LIN {X -0.158,Y -481.515,Z 1004.070,A 0.000,B 0.000,C 90.000,E1 228.528} C_DIS
LIN {X -0.055,Y -475.509,Z 1004.054,A 0.000,B 0.000,C 90.000,E1 225.729} C_DIS
LIN {X -0.116,Y -471.668,Z 1004.044,A 0.000,B 0.000,C 90.000,E1 223.866} C_DIS
LIN {X -0.012,Y -468.320,Z 1004.035,A 0.000,B 0.000,C 90.000,E1 222.285} C_DIS
LIN {X 0.118,Y -464.188,Z 1004.024,A 0.000,B 0.000,C 90.000,E1 220.378} C_DIS
LIN {X 0.208,Y -459.845,Z 1004.014,A 0.000,B 0.000,C 90.000,E1 218.463} C_DIS
LIN {X -0.083,Y -455.698,Z 1004.003,A 0.000,B 0.000,C 90.000,E1 216.583} C_DIS
LIN {X 0.261,Y -451.461,Z 1003.992,A 0.000,B 0.000,C 90.000,E1 214.612} C_DIS
LIN {X 0.003,Y -447.260,Z 1003.982,A 0.000,B 0.000,C 90.000,E1 212.704} C_DIS
LIN {X -0.029,Y -443.708,Z 1003.973,A 0.000,B 0.000,C 90.000,E1 211.082} C_DIS
LIN {X -0.140,Y -440.143,Z 1003.964,A 0.000,B 0.000,C 90.000,E1 209.461} C_DIS
LIN {X 0.041,Y -435.600,Z 1003.953,A 0.000,B 0.000,C 90.000,E1 207.462} C_DIS
LIN {X 0.115,Y -431.912,Z 1003.943,A 0.000,B 0.000,C 90.000,E1 205.796} C_DIS
LIN {X 0.105,Y -428.119,Z 1003.934,A 0.000,B 0.000,C 90.000,E1 204.131} C_DIS
LIN {X -0.147,Y -423.631,Z 1003.923,A 0.000,B 0.000,C 90.000,E1 202.153} C_DIS
LIN {X -0.164,Y -417.964,Z 1003.908,A 0.000,B 0.000,C 90.000,E1 199.450} C_DIS
LIN {X -0.090,Y -411.609,Z 1003.889,A 0.000,B 0.000,C 90.000,E1 196.024} C_DIS
LIN {X -0.066,Y -408.697,Z 1003.879,A 0.000,B 0.000,C 90.000,E1 194.300} C_DIS
LIN {X 0.193,Y -405.963,Z 1003.870,A 0.000,B 0.000,C 90.000,E1 192.535} C_DIS
LIN {X -0.085,Y -403.341,Z 1003.860,A 0.000,B 0.000,C 90.000,E1 190.838} C_DIS
LIN {X -0.083,Y -401.810,Z 1003.854,A 0.000,B 0.000,C 90.000,E1 189.792} C_DIS
LIN {X -0.106,Y -400.288,Z 1003.847,A 0.000,B 0.000,C 90.000,E1 188.398} C_DIS
LIN {X -0.144,Y -400.025,Z 1003.841,A 0.000,B 0.000,C 90.000,E1 187.352} C_DIS
LIN {X -0.116,Y -400.167,Z 1003.839,A 0.000,B 0.000,C 90.000,E1 187.004} C_DIS
LIN {X 0.119,Y -400.532,Z 1003.838,A 0.000,B 0.000,C 90.000,E1 186.777} C_DIS
LIN {X 0.045,Y -401.446,Z 1003.834,A 0.000,B 0.000,C 90.000,E1 186.087} C_DIS
LIN {X 0.019,Y -402.755,Z 1003.831,A 0.000,B 0.000,C 90.000,E1 185.568} C_DIS
LIN {X 0.143,Y -405.533,Z 1003.827,A 0.000,B 0.000,C 90.000,E1 184.878} C_DIS
LIN {X 0.140,Y -407.318,Z 1003.825,A 0.000,B 0.000,C 90.000,E1 184.531} C_DIS
LIN {X 0.080,Y -410.355,Z 1003.823,A 0.000,B 0.000,C 90.000,E1 184.073} C_DIS
LIN {X 0.140,Y -415.263,Z 1003.819,A 0.000,B 0.000,C 90.000,E1 183.440} C_DIS
LIN {X -0.203,Y -423.575,Z 1003.814,A 0.000,B 0.000,C 90.000,E1 182.522} C_DIS
LIN {X -0.028,Y -430.671,Z 1003.810,A 0.000,B 0.000,C 90.000,E1 181.718} C_DIS
LIN {X 0.109,Y -442.868,Z 1003.802,A 0.000,B 0.000,C 90.000,E1 180.344} C_DIS
LIN {X 0.157,Y -455.130,Z 1003.794,A 0.000,B 0.000,C 90.000,E1 178.969} C_DIS
LIN {X 0.082,Y -463.200,Z 1003.789,A 0.000,B 0.000,C 90.000,E1 178.051} C_DIS
LIN {X 0.169,Y -468.505,Z 1003.786,A 0.000,B 0.000,C 90.000,E1 177.421} C_DIS
LIN {X 0.143,Y -476.033,Z 1003.781,A 0.000,B 0.000,C 90.000,E1 176.502} C_DIS
LIN {X -0.110,Y -482.206,Z 1003.776,A 0.000,B 0.000,C 90.000,E1 175.755} C_DIS
LIN {X 0.000,Y -490.150,Z 1003.770,A 0.000,B 0.000,C 90.000,E1 174.666} C_DIS
LIN {X 0.089,Y -496.507,Z 1003.765,A 0.000,B 0.000,C 90.000,E1 173.742} C_DIS
LIN {X 0.009,Y -503.705,Z 1003.760,A 0.000,B 0.000,C 90.000,E1 172.704} C_DIS
LIN {X -0.213,Y -511.598,Z 1003.753,A 0.000,B 0.000,C 90.000,E1 171.546} C_DIS
LIN {X -0.104,Y -519.992,Z 1003.746,A 0.000,B 0.000,C 90.000,E1 170.208} C_DIS
LIN {X 0.120,Y -526.038,Z 1003.740,A 0.000,B 0.000,C 90.000,E1 169.162} C_DIS
LIN {X -0.160,Y -528.740,Z 1003.737,A 0.000,B 0.000,C 90.000,E1 168.757} C_DIS
LIN {X 0.215,Y -538.987,Z 1003.728,A 0.000,B 0.000,C 90.000,E1 166.992} C_DIS
LIN {X 0.272,Y -544.731,Z 1003.722,A 0.000,B 0.000,C 90.000,E1 165.992} C_DIS
LIN {X 0.014,Y -549.638,Z 1003.718,A 0.000,B 0.000,C 90.000,E1 165.172} C_DIS
LIN {X -0.192,Y -555.149,Z 1003.712,A 0.000,B 0.000,C 90.000,E1 164.212} C_DIS
LIN {X -0.191,Y -561.923,Z 1003.705,A 0.000,B 0.000,C 90.000,E1 162.960} C_DIS
LIN {X 0.244,Y -569.849,Z 1003.697,A 0.000,B 0.000,C 90.000,E1 161.402} C_DIS
LIN {X -0.065,Y -574.593,Z 1003.692,A 0.000,B 0.000,C 90.000,E1 160.477} C_DIS
LIN {X 0.112,Y -578.574,Z 1003.687,A 0.000,B 0.000,C 90.000,E1 159.645} C_DIS
LIN {X -0.089,Y -582.935,Z 1003.682,A 0.000,B 0.000,C 90.000,E1 158.720} C_DIS
LIN {X 0.111,Y -586.015,Z 1003.678,A 0.000,B 0.000,C 90.000,E1 158.028} C_DIS
LIN {X -0.060,Y -590.629,Z 1003.672,A 0.000,B 0.000,C 90.000,E1 156.975} C_DIS
LIN {X -0.174,Y -594.836,Z 1003.666,A 0.000,B 0.000,C 90.000,E1 155.921} C_DIS
LIN {X 0.009,Y -598.632,Z 1003.660,A 0.000,B 0.000,C 90.000,E1 154.845} C_DIS
LIN {X 0.319,Y -601.320,Z 1003.656,A 0.000,B 0.000,C 90.000,E1 154.024} C_DIS
LIN {X 0.052,Y -604.541,Z 1003.650,A 0.000,B 0.000,C 90.000,E1 152.999} C_DIS
LIN {X 0.011,Y -609.120,Z 1003.641,A 0.000,B 0.000,C 90.000,E1 151.435} C_DIS
LIN {X 0.062,Y -613.469,Z 1003.633,A 0.000,B 0.000,C 90.000,E1 149.871} C_DIS
LIN {X -0.290,Y -616.337,Z 1003.627,A 0.000,B 0.000,C 90.000,E1 148.869} C_DIS
LIN {X 0.222,Y -619.799,Z 1003.620,A 0.000,B 0.000,C 90.000,E1 147.533} C_DIS
LIN {X 0.054,Y -624.612,Z 1003.610,A 0.000,B 0.000,C 90.000,E1 145.754} C_DIS
LIN {X -0.164,Y -629.479,Z 1003.600,A 0.000,B 0.000,C 90.000,E1 143.989} C_DIS
LIN {X -0.261,Y -633.516,Z 1003.591,A 0.000,B 0.000,C 90.000,E1 142.477} C_DIS
LIN {X 0.234,Y -636.871,Z 1003.584,A 0.000,B 0.000,C 90.000,E1 141.170} C_DIS
LIN {X 0.289,Y -640.156,Z 1003.577,A 0.000,B 0.000,C 90.000,E1 139.908} C_DIS
LIN {X -0.007,Y -642.774,Z 1003.572,A 0.000,B 0.000,C 90.000,E1 138.933} C_DIS
LIN {X -0.084,Y -647.947,Z 1003.561,A 0.000,B 0.000,C 90.000,E1 136.944} C_DIS
LIN {X 0.037,Y -652.110,Z 1003.553,A 0.000,B 0.000,C 90.000,E1 135.445} C_DIS
LIN {X 0.114,Y -659.741,Z 1003.539,A 0.000,B 0.000,C 90.000,E1 132.975} C_DIS
LIN {X 0.065,Y -666.201,Z 1003.528,A 0.000,B 0.000,C 90.000,E1 131.024} C_DIS
LIN {X -0.397,Y -669.403,Z 1003.523,A 0.000,B 0.000,C 90.000,E1 130.092} C_DIS
LIN {X -0.316,Y -672.466,Z 1003.517,A 0.000,B 0.000,C 90.000,E1 129.116} C_DIS
LIN {X -0.082,Y -675.979,Z 1003.510,A 0.000,B 0.000,C 90.000,E1 127.890} C_DIS
LIN {X -0.176,Y -680.134,Z 1003.503,A 0.000,B 0.000,C 90.000,E1 126.457} C_DIS
LIN {X -0.198,Y -684.071,Z 1003.495,A 0.000,B 0.000,C 90.000,E1 125.025} C_DIS
LIN {X -0.181,Y -687.276,Z 1003.488,A 0.000,B 0.000,C 90.000,E1 123.833} C_DIS
LIN {X 0.235,Y -689.124,Z 1003.484,A 0.000,B 0.000,C 90.000,E1 123.086} C_DIS
LIN {X 0.178,Y -692.714,Z 1003.476,A 0.000,B 0.000,C 90.000,E1 121.671} C_DIS
LIN {X -0.059,Y -695.075,Z 1003.471,A 0.000,B 0.000,C 90.000,E1 120.747} C_DIS
LIN {X -0.166,Y -696.680,Z 1003.467,A 0.000,B 0.000,C 90.000,E1 120.050} C_DIS
LIN {X 0.341,Y -697.649,Z 1003.464,A 0.000,B 0.000,C 90.000,E1 119.539} C_DIS
LIN {X 0.163,Y -699.184,Z 1003.459,A 0.000,B 0.000,C 90.000,E1 118.615} C_DIS
LIN {X -0.328,Y -700.404,Z 1003.454,A 0.000,B 0.000,C 90.000,E1 117.719} C_DIS
LIN {X -0.324,Y -701.880,Z 1003.443,A 0.000,B 0.000,C 90.000,E1 115.848} C_DIS
LIN {X -0.149,Y -702.550,Z 1003.438,A 0.000,B 0.000,C 90.000,E1 114.899} C_DIS
LIN {X -0.244,Y -702.705,Z 1003.434,A 0.000,B 0.000,C 90.000,E1 114.207} C_DIS
LIN {X 0.310,Y -702.127,Z 1003.432,A 0.000,B 0.000,C 90.000,E1 113.695} C_DIS
LIN {X -0.339,Y -701.687,Z 1003.431,A 0.000,B 0.000,C 90.000,E1 113.515} C_DIS
LIN {X 0.065,Y -699.072,Z 1003.427,A 0.000,B 0.000,C 90.000,E1 112.898} C_DIS
LIN {X 0.199,Y -698.300,Z 1003.427,A 0.000,B 0.000,C 90.000,E1 112.770} C_DIS
LIN {X 0.328,Y -697.150,Z 1003.426,A 0.000,B 0.000,C 90.000,E1 112.642} C_DIS
LIN {X 0.151,Y -692.817,Z 1003.424,A 0.000,B 0.000,C 90.000,E1 112.333} C_DIS
LIN {X -0.159,Y -691.331,Z 1003.424,A 0.000,B 0.000,C 90.000,E1 112.259} C_DIS
LIN {X -0.092,Y -689.495,Z 1003.423,A 0.000,B 0.000,C 90.000,E1 112.153} C_DIS
LIN {X 0.058,Y -684.547,Z 1003.422,A 0.000,B 0.000,C 90.000,E1 111.972} C_DIS
LIN {X 0.216,Y -677.312,Z 1003.422,A 0.000,B 0.000,C 90.000,E1 111.844} C_DIS
LIN {X -0.113,Y -675.141,Z 1003.421,A 0.000,B 0.000,C 90.000,E1 111.844} C_DIS
LIN {X -0.164,Y -669.455,Z 1003.421,A 0.000,B 0.000,C 90.000,E1 111.844} C_DIS
LIN {X -0.198,Y -618.340,Z 1003.421,A 0.000,B 0.000,C 90.000,E1 111.844} C_DIS
LIN {X -0.208,Y -614.996,Z 1003.421,A 0.000,B 0.000,C 90.000,E1 111.770} C_DIS
LIN {X -0.025,Y -610.858,Z 1003.420,A 0.000,B 0.000,C 90.000,E1 111.642} C_DIS
LIN {X -0.146,Y -604.502,Z 1003.419,A 0.000,B 0.000,C 90.000,E1 111.408} C_DIS
LIN {X -0.108,Y -601.661,Z 1003.418,A 0.000,B 0.000,C 90.000,E1 111.280} C_DIS
LIN {X -0.047,Y -595.162,Z 1003.416,A 0.000,B 0.000,C 90.000,E1 110.918} C_DIS
LIN {X 0.031,Y -589.063,Z 1003.414,A 0.000,B 0.000,C 90.000,E1 110.482} C_DIS
LIN {X 0.107,Y -577.100,Z 1003.408,A 0.000,B 0.000,C 90.000,E1 109.504} C_DIS
LIN {X 0.298,Y -572.724,Z 1003.407,A 0.000,B 0.000,C 90.000,E1 109.141} C_DIS
LIN {X -0.084,Y -564.162,Z 1003.404,A 0.000,B 0.000,C 90.000,E1 108.671} C_DIS
LIN {X 0.140,Y -550.287,Z 1003.400,A 0.000,B 0.000,C 90.000,E1 107.946} C_DIS
LIN {X -0.224,Y -548.864,Z 1003.399,A 0.000,B 0.000,C 90.000,E1 107.819} C_DIS
LIN {X -0.266,Y -548.850,Z 1003.399,A 0.000,B 0.000,C 90.000,E1 107.819} C_DIS
LIN {X -0.134,Y -548.453,Z 1003.397,A 0.000,B 0.000,C 90.000,E1 107.511} C_DIS
LIN {X -0.090,Y -548.522,Z 1003.393,A 0.000,B 0.000,C 90.000,E1 106.804} C_DIS
LIN {X 0.171,Y -549.154,Z 1003.386,A 0.000,B 0.000,C 90.000,E1 105.371} C_DIS
LIN {X 0.220,Y -550.329,Z 1003.373,A 0.000,B 0.000,C 90.000,E1 103.119} C_DIS
LIN {X 0.288,Y -552.781,Z 1003.357,A 0.000,B 0.000,C 90.000,E1 100.310} C_DIS
LIN {X -0.130,Y -554.939,Z 1003.347,A 0.000,B 0.000,C 90.000,E1 98.398} C_DIS
LIN {X -0.133,Y -556.428,Z 1003.339,A 0.000,B 0.000,C 90.000,E1 97.004} C_DIS
LIN {X -0.246,Y -557.751,Z 1003.331,A 0.000,B 0.000,C 90.000,E1 95.625} C_DIS
LIN {X 0.230,Y -558.784,Z 1003.323,A 0.000,B 0.000,C 90.000,E1 94.188} C_DIS
LIN {X 0.162,Y -559.630,Z 1003.316,A 0.000,B 0.000,C 90.000,E1 92.808} C_DIS
LIN {X -0.209,Y -560.695,Z 1003.303,A 0.000,B 0.000,C 90.000,E1 90.630} C_DIS
LIN {X 0.174,Y -561.210,Z 1003.297,A 0.000,B 0.000,C 90.000,E1 89.484} C_DIS
LIN {X 0.115,Y -561.773,Z 1003.290,A 0.000,B 0.000,C 90.000,E1 88.108} C_DIS
LIN {X 0.069,Y -562.004,Z 1003.282,A 0.000,B 0.000,C 90.000,E1 86.731} C_DIS
LIN {X -0.073,Y -562.162,Z 1003.276,A 0.000,B 0.000,C 90.000,E1 85.641} C_DIS
LIN {X -0.082,Y -562.395,Z 1003.268,A 0.000,B 0.000,C 90.000,E1 84.261} C_DIS
LIN {X 0.204,Y -562.712,Z 1003.257,A 0.000,B 0.000,C 90.000,E1 82.299} C_DIS
LIN {X -0.142,Y -563.152,Z 1003.248,A 0.000,B 0.000,C 90.000,E1 80.679} C_DIS
LIN {X -0.228,Y -563.904,Z 1003.237,A 0.000,B 0.000,C 90.000,E1 78.757} C_DIS
LIN {X 0.201,Y -564.750,Z 1003.228,A 0.000,B 0.000,C 90.000,E1 77.061} C_DIS
LIN {X 0.221,Y -565.722,Z 1003.219,A 0.000,B 0.000,C 90.000,E1 75.408} C_DIS
LIN {X -0.129,Y -566.892,Z 1003.210,A 0.000,B 0.000,C 90.000,E1 73.795} C_DIS
LIN {X -0.116,Y -568.379,Z 1003.199,A 0.000,B 0.000,C 90.000,E1 71.873} C_DIS
LIN {X 0.110,Y -569.709,Z 1003.189,A 0.000,B 0.000,C 90.000,E1 69.934} C_DIS
LIN {X 0.206,Y -570.687,Z 1003.180,A 0.000,B 0.000,C 90.000,E1 68.284} C_DIS
LIN {X 0.171,Y -571.364,Z 1003.172,A 0.000,B 0.000,C 90.000,E1 66.922} C_DIS
LIN {X 0.021,Y -571.901,Z 1003.166,A 0.000,B 0.000,C 90.000,E1 65.845} C_DIS
LIN {X 0.076,Y -572.579,Z 1003.157,A 0.000,B 0.000,C 90.000,E1 64.204} C_DIS
LIN {X 0.129,Y -573.079,Z 1003.148,A 0.000,B 0.000,C 90.000,E1 62.564} C_DIS
LIN {X 0.366,Y -573.489,Z 1003.140,A 0.000,B 0.000,C 90.000,E1 61.179} C_DIS
LIN {X -0.162,Y -573.872,Z 1003.133,A 0.000,B 0.000,C 90.000,E1 59.871} C_DIS
LIN {X 0.089,Y -574.151,Z 1003.125,A 0.000,B 0.000,C 90.000,E1 58.486} C_DIS
LIN {X 0.018,Y -574.306,Z 1003.119,A 0.000,B 0.000,C 90.000,E1 57.406} C_DIS
LIN {X -0.248,Y -574.580,Z 1003.110,A 0.000,B 0.000,C 90.000,E1 55.801} C_DIS
LIN {X 0.007,Y -574.612,Z 1003.104,A 0.000,B 0.000,C 90.000,E1 54.689} C_DIS
LIN {X -0.058,Y -574.439,Z 1003.096,A 0.000,B 0.000,C 90.000,E1 53.336} C_DIS
LIN {X 0.036,Y -574.222,Z 1003.092,A 0.000,B 0.000,C 90.000,E1 52.512} C_DIS
LIN {X 0.159,Y -573.718,Z 1003.086,A 0.000,B 0.000,C 90.000,E1 51.412} C_DIS
LIN {X -0.027,Y -572.906,Z 1003.078,A 0.000,B 0.000,C 90.000,E1 50.070} C_DIS
LIN {X 0.148,Y -571.824,Z 1003.071,A 0.000,B 0.000,C 90.000,E1 48.690} C_DIS
LIN {X -0.200,Y -570.727,Z 1003.065,A 0.000,B 0.000,C 90.000,E1 47.634} C_DIS
LIN {X 0.120,Y -569.705,Z 1003.060,A 0.000,B 0.000,C 90.000,E1 46.782} C_DIS
LIN {X 0.016,Y -568.470,Z 1003.055,A 0.000,B 0.000,C 90.000,E1 45.972} C_DIS
LIN {X -0.098,Y -567.024,Z 1003.051,A 0.000,B 0.000,C 90.000,E1 45.162} C_DIS
LIN {X -0.225,Y -565.417,Z 1003.046,A 0.000,B 0.000,C 90.000,E1 44.352} C_DIS
LIN {X 0.106,Y -563.058,Z 1003.040,A 0.000,B 0.000,C 90.000,E1 43.218} C_DIS
LIN {X -0.038,Y -560.958,Z 1003.036,A 0.000,B 0.000,C 90.000,E1 42.405} C_DIS
LIN {X -0.238,Y -558.549,Z 1003.031,A 0.000,B 0.000,C 90.000,E1 41.595} C_DIS
LIN {X -0.054,Y -555.831,Z 1003.026,A 0.000,B 0.000,C 90.000,E1 40.744} C_DIS
LIN {X 0.092,Y -553.882,Z 1003.023,A 0.000,B 0.000,C 90.000,E1 40.172} C_DIS
LIN {X -0.195,Y -551.798,Z 1003.020,A 0.000,B 0.000,C 90.000,E1 39.644} C_DIS
LIN {X 0.132,Y -548.920,Z 1003.016,A 0.000,B 0.000,C 90.000,E1 38.910} C_DIS
LIN {X -0.107,Y -543.889,Z 1003.010,A 0.000,B 0.000,C 90.000,E1 37.810} C_DIS
LIN {X -0.014,Y -539.741,Z 1003.005,A 0.000,B 0.000,C 90.000,E1 36.950} C_DIS
LIN {X 0.035,Y -535.405,Z 1003.001,A 0.000,B 0.000,C 90.000,E1 36.091} C_DIS
LIN {X 0.033,Y -530.741,Z 1002.996,A 0.000,B 0.000,C 90.000,E1 35.231} C_DIS
LIN {X -0.160,Y -526.639,Z 1002.992,A 0.000,B 0.000,C 90.000,E1 34.532} C_DIS
LIN {X -0.123,Y -521.403,Z 1002.987,A 0.000,B 0.000,C 90.000,E1 33.658} C_DIS
LIN {X 0.036,Y -516.696,Z 1002.983,A 0.000,B 0.000,C 90.000,E1 32.911} C_DIS
LIN {X -0.280,Y -511.671,Z 1002.979,A 0.000,B 0.000,C 90.000,E1 32.212} C_DIS
LIN {X -0.214,Y -506.316,Z 1002.975,A 0.000,B 0.000,C 90.000,E1 31.465} C_DIS
LIN {X -0.137,Y -501.769,Z 1002.971,A 0.000,B 0.000,C 90.000,E1 30.875} C_DIS
LIN {X 0.031,Y -496.671,Z 1002.968,A 0.000,B 0.000,C 90.000,E1 30.256} C_DIS
LIN {X 0.021,Y -491.298,Z 1002.965,A 0.000,B 0.000,C 90.000,E1 29.667} C_DIS
LIN {X -0.060,Y -484.415,Z 1002.961,A 0.000,B 0.000,C 90.000,E1 28.949} C_DIS
LIN {X -0.009,Y -475.815,Z 1002.956,A 0.000,B 0.000,C 90.000,E1 28.103} C_DIS
LIN {X 0.220,Y -467.202,Z 1002.952,A 0.000,B 0.000,C 90.000,E1 27.257} C_DIS
LIN {X -0.024,Y -458.276,Z 1002.947,A 0.000,B 0.000,C 90.000,E1 26.488} C_DIS
LIN {X -0.192,Y -449.137,Z 1002.943,A 0.000,B 0.000,C 90.000,E1 25.720} C_DIS
LIN {X -0.076,Y -428.087,Z 1002.933,A 0.000,B 0.000,C 90.000,E1 23.875} C_DIS
LIN {X -0.047,Y -414.723,Z 1002.926,A 0.000,B 0.000,C 90.000,E1 22.589} C_DIS
LIN {X 0.147,Y -400.598,Z 1002.917,A 0.000,B 0.000,C 90.000,E1 21.046} C_DIS
LIN {X 0.084,Y -397.931,Z 1002.915,A 0.000,B 0.000,C 90.000,E1 20.737} C_DIS
LIN {X -0.101,Y -394.399,Z 1002.912,A 0.000,B 0.000,C 90.000,E1 20.248} C_DIS
LIN {X 0.005,Y -391.847,Z 1002.909,A 0.000,B 0.000,C 90.000,E1 19.685} C_DIS
LIN {X 0.080,Y -390.658,Z 1002.906,A 0.000,B 0.000,C 90.000,E1 19.141} C_DIS
LIN {X -0.090,Y -390.421,Z 1002.903,A 0.000,B 0.000,C 90.000,E1 18.544} C_DIS
LIN {X -0.183,Y -391.164,Z 1002.897,A 0.000,B 0.000,C 90.000,E1 17.457} C_DIS
LIN {X -0.021,Y -394.023,Z 1002.881,A 0.000,B 0.000,C 90.000,E1 14.592} C_DIS
LIN {X -0.053,Y -399.154,Z 1002.860,A 0.000,B 0.000,C 90.000,E1 10.715} C_DIS
LIN {X 0.198,Y -405.816,Z 1002.838,A 0.000,B 0.000,C 90.000,E1 6.834} C_DIS
LIN {X 0.161,Y -412.315,Z 1002.821,A 0.000,B 0.000,C 90.000,E1 3.726} C_DIS
LIN {X -0.191,Y -416.990,Z 1002.809,A 0.000,B 0.000,C 90.000,E1 1.718} C_DIS
LIN {X -0.155,Y -419.463,Z 1002.806,A 0.000,B 0.000,C 90.000,E1 1.031} C_DIS
LIN {X 0.104,Y -422.290,Z 1002.803,A 0.000,B 0.000,C 90.000,E1 0.516} C_DIS
LIN {X 0.121,Y -423.471,Z 1002.802,A 0.000,B 0.000,C 90.000,E1 0.344} C_DIS
LIN {X 0.081,Y -428.417,Z 1002.799,A 0.000,B 0.000,C 90.000,E1 359.885} C_DIS
LIN {X -0.081,Y -435.391,Z 1002.797,A 0.000,B 0.000,C 90.000,E1 359.484} C_DIS
LIN {X 0.058,Y -443.314,Z 1002.795,A 0.000,B 0.000,C 90.000,E1 359.026} C_DIS
LIN {X -0.103,Y -456.708,Z 1002.790,A 0.000,B 0.000,C 90.000,E1 358.282} C_DIS
LIN {X -0.140,Y -466.697,Z 1002.787,A 0.000,B 0.000,C 90.000,E1 357.707} C_DIS
LIN {X 0.001,Y -483.324,Z 1002.782,A 0.000,B 0.000,C 90.000,E1 356.731} C_DIS
LIN {X 0.101,Y -493.014,Z 1002.779,A 0.000,B 0.000,C 90.000,E1 356.159} C_DIS
LIN {X -0.027,Y -505.539,Z 1002.775,A 0.000,B 0.000,C 90.000,E1 355.412} C_DIS
LIN {X -0.007,Y -510.206,Z 1002.773,A 0.000,B 0.000,C 90.000,E1 355.122} C_DIS
LIN {X -0.049,Y -517.751,Z 1002.770,A 0.000,B 0.000,C 90.000,E1 354.609} C_DIS
LIN {X 0.124,Y -525.283,Z 1002.767,A 0.000,B 0.000,C 90.000,E1 354.033} C_DIS
LIN {X 0.228,Y -532.376,Z 1002.764,A 0.000,B 0.000,C 90.000,E1 353.457} C_DIS
LIN {X 0.006,Y -538.031,Z 1002.761,A 0.000,B 0.000,C 90.000,E1 352.996} C_DIS
LIN {X 0.252,Y -543.439,Z 1002.758,A 0.000,B 0.000,C 90.000,E1 352.470} C_DIS
LIN {X 0.032,Y -549.815,Z 1002.755,A 0.000,B 0.000,C 90.000,E1 351.837} C_DIS
LIN {X -0.191,Y -554.829,Z 1002.752,A 0.000,B 0.000,C 90.000,E1 351.310} C_DIS
LIN {X -0.276,Y -560.507,Z 1002.748,A 0.000,B 0.000,C 90.000,E1 350.622} C_DIS
LIN {X 0.269,Y -563.734,Z 1002.745,A 0.000,B 0.000,C 90.000,E1 350.151} C_DIS
LIN {X -0.203,Y -568.380,Z 1002.742,A 0.000,B 0.000,C 90.000,E1 349.511} C_DIS
LIN {X -0.081,Y -572.570,Z 1002.738,A 0.000,B 0.000,C 90.000,E1 348.814} C_DIS
LIN {X -0.249,Y -575.735,Z 1002.735,A 0.000,B 0.000,C 90.000,E1 348.285} C_DIS
LIN {X 0.153,Y -580.883,Z 1002.730,A 0.000,B 0.000,C 90.000,E1 347.297} C_DIS
LIN {X -0.152,Y -586.941,Z 1002.723,A 0.000,B 0.000,C 90.000,E1 346.117} C_DIS
LIN {X -0.135,Y -592.014,Z 1002.717,A 0.000,B 0.000,C 90.000,E1 345.046} C_DIS
LIN {X -0.048,Y -596.791,Z 1002.711,A 0.000,B 0.000,C 90.000,E1 343.976} C_DIS
LIN {X -0.185,Y -602.327,Z 1002.704,A 0.000,B 0.000,C 90.000,E1 342.670} C_DIS
LIN {X 0.213,Y -606.500,Z 1002.698,A 0.000,B 0.000,C 90.000,E1 341.583} C_DIS
LIN {X 0.100,Y -610.483,Z 1002.692,A 0.000,B 0.000,C 90.000,E1 340.550} C_DIS
LIN {X -0.226,Y -612.453,Z 1002.689,A 0.000,B 0.000,C 90.000,E1 340.061} C_DIS
LIN {X -0.263,Y -615.854,Z 1002.683,A 0.000,B 0.000,C 90.000,E1 339.028} C_DIS
LIN {X 0.252,Y -621.319,Z 1002.673,A 0.000,B 0.000,C 90.000,E1 337.177} C_DIS
LIN {X -0.016,Y -624.203,Z 1002.668,A 0.000,B 0.000,C 90.000,E1 336.177} C_DIS
LIN {X -0.236,Y -627.442,Z 1002.661,A 0.000,B 0.000,C 90.000,E1 334.921} C_DIS
LIN {X -0.158,Y -629.879,Z 1002.655,A 0.000,B 0.000,C 90.000,E1 333.896} C_DIS
LIN {X -0.075,Y -631.565,Z 1002.651,A 0.000,B 0.000,C 90.000,E1 333.127} C_DIS
LIN {X 0.095,Y -633.990,Z 1002.644,A 0.000,B 0.000,C 90.000,E1 331.847} C_DIS
LIN {X -0.038,Y -635.383,Z 1002.639,A 0.000,B 0.000,C 90.000,E1 331.101} C_DIS
LIN {X -0.369,Y -637.535,Z 1002.633,A 0.000,B 0.000,C 90.000,E1 329.871} C_DIS
LIN {X -0.025,Y -639.507,Z 1002.625,A 0.000,B 0.000,C 90.000,E1 328.584} C_DIS
LIN {X -0.032,Y -640.805,Z 1002.620,A 0.000,B 0.000,C 90.000,E1 327.582} C_DIS
LIN {X -0.032,Y -641.962,Z 1002.614,A 0.000,B 0.000,C 90.000,E1 326.580} C_DIS
LIN {X 0.285,Y -642.719,Z 1002.610,A 0.000,B 0.000,C 90.000,E1 325.801} C_DIS
LIN {X 0.134,Y -643.596,Z 1002.605,A 0.000,B 0.000,C 90.000,E1 324.815} C_DIS
LIN {X 0.030,Y -644.280,Z 1002.598,A 0.000,B 0.000,C 90.000,E1 323.577} C_DIS
LIN {X 0.210,Y -644.967,Z 1002.589,A 0.000,B 0.000,C 90.000,E1 322.065} C_DIS
LIN {X -0.107,Y -645.471,Z 1002.581,A 0.000,B 0.000,C 90.000,E1 320.598} C_DIS
LIN {X 0.268,Y -646.386,Z 1002.569,A 0.000,B 0.000,C 90.000,E1 318.324} C_DIS
LIN {X -0.027,Y -647.218,Z 1002.562,A 0.000,B 0.000,C 90.000,E1 317.106} C_DIS
LIN {X -0.001,Y -648.187,Z 1002.552,A 0.000,B 0.000,C 90.000,E1 315.364} C_DIS
LIN {X 0.051,Y -649.286,Z 1002.542,A 0.000,B 0.000,C 90.000,E1 313.623} C_DIS
LIN {X 0.243,Y -650.142,Z 1002.536,A 0.000,B 0.000,C 90.000,E1 312.366} C_DIS
LIN {X 0.070,Y -650.746,Z 1002.530,A 0.000,B 0.000,C 90.000,E1 311.391} C_DIS
LIN {X -0.147,Y -651.458,Z 1002.523,A 0.000,B 0.000,C 90.000,E1 310.172} C_DIS
LIN {X -0.391,Y -652.190,Z 1002.514,A 0.000,B 0.000,C 90.000,E1 308.463} C_DIS
LIN {X -0.099,Y -652.636,Z 1002.507,A 0.000,B 0.000,C 90.000,E1 307.202} C_DIS
LIN {X -0.056,Y -652.850,Z 1002.503,A 0.000,B 0.000,C 90.000,E1 306.457} C_DIS
LIN {X -0.080,Y -653.067,Z 1002.494,A 0.000,B 0.000,C 90.000,E1 304.978} C_DIS
LIN {X -0.020,Y -653.472,Z 1002.485,A 0.000,B 0.000,C 90.000,E1 303.245} C_DIS
LIN {X -0.373,Y -657.762,Z 1002.456,A 0.000,B 0.000,C 90.000,E1 298.103} C_DIS
LIN {X -0.209,Y -659.767,Z 1002.448,A 0.000,B 0.000,C 90.000,E1 296.616} C_DIS
LIN {X -0.300,Y -661.870,Z 1002.440,A 0.000,B 0.000,C 90.000,E1 295.155} C_DIS
LIN {X 0.111,Y -663.327,Z 1002.433,A 0.000,B 0.000,C 90.000,E1 293.898} C_DIS
LIN {X -0.207,Y -664.099,Z 1002.427,A 0.000,B 0.000,C 90.000,E1 292.950} C_DIS
LIN {X -0.187,Y -664.362,Z 1002.425,A 0.000,B 0.000,C 90.000,E1 292.461} C_DIS
LIN {X -0.162,Y -664.413,Z 1002.422,A 0.000,B 0.000,C 90.000,E1 291.972} C_DIS
LIN {X 0.109,Y -664.021,Z 1002.419,A 0.000,B 0.000,C 90.000,E1 291.461} C_DIS
LIN {X 0.000,Y -663.557,Z 1002.418,A 0.000,B 0.000,C 90.000,E1 291.227} C_DIS
LIN {X 0.131,Y -662.899,Z 1002.417,A 0.000,B 0.000,C 90.000,E1 290.972} C_DIS
LIN {X 0.024,Y -662.003,Z 1002.415,A 0.000,B 0.000,C 90.000,E1 290.737} C_DIS
LIN {X 0.086,Y -661.351,Z 1002.415,A 0.000,B 0.000,C 90.000,E1 290.610} C_DIS
LIN {X 0.036,Y -658.734,Z 1002.413,A 0.000,B 0.000,C 90.000,E1 290.248} C_DIS
LIN {X 0.092,Y -657.656,Z 1002.412,A 0.000,B 0.000,C 90.000,E1 290.120} C_DIS
LIN {X 0.146,Y -656.396,Z 1002.411,A 0.000,B 0.000,C 90.000,E1 289.993} C_DIS
LIN {X 0.009,Y -654.777,Z 1002.411,A 0.000,B 0.000,C 90.000,E1 289.885} C_DIS
LIN {X -0.245,Y -648.371,Z 1002.408,A 0.000,B 0.000,C 90.000,E1 289.504} C_DIS
LIN {X -0.267,Y -637.490,Z 1002.405,A 0.000,B 0.000,C 90.000,E1 288.906} C_DIS
LIN {X -0.332,Y -637.406,Z 1002.405,A 0.000,B 0.000,C 90.000,E1 288.906} C_DIS
LIN {X -0.103,Y -636.148,Z 1002.404,A 0.000,B 0.000,C 90.000,E1 288.725} C_DIS
LIN {X -0.147,Y -636.131,Z 1002.404,A 0.000,B 0.000,C 90.000,E1 288.725} C_DIS
LIN {X -0.020,Y -636.406,Z 1002.403,A 0.000,B 0.000,C 90.000,E1 288.489} C_DIS
LIN {X -0.310,Y -640.874,Z 1002.399,A 0.000,B 0.000,C 90.000,E1 287.764} C_DIS
LIN {X 0.210,Y -644.114,Z 1002.396,A 0.000,B 0.000,C 90.000,E1 287.221} C_DIS
LIN {X -0.028,Y -647.825,Z 1002.392,A 0.000,B 0.000,C 90.000,E1 286.622} C_DIS
LIN {X -0.260,Y -651.699,Z 1002.388,A 0.000,B 0.000,C 90.000,E1 285.898} C_DIS
LIN {X 0.114,Y -653.709,Z 1002.385,A 0.000,B 0.000,C 90.000,E1 285.371} C_DIS
LIN {X -0.009,Y -654.617,Z 1002.384,A 0.000,B 0.000,C 90.000,E1 285.134} C_DIS
LIN {X -0.077,Y -656.169,Z 1002.381,A 0.000,B 0.000,C 90.000,E1 284.647} C_DIS
LIN {X 0.331,Y -657.306,Z 1002.379,A 0.000,B 0.000,C 90.000,E1 284.120} C_DIS
LIN {X 0.006,Y -658.605,Z 1002.375,A 0.000,B 0.000,C 90.000,E1 283.411} C_DIS
LIN {X 0.332,Y -659.271,Z 1002.370,A 0.000,B 0.000,C 90.000,E1 282.647} C_DIS
LIN {X -0.015,Y -659.435,Z 1002.368,A 0.000,B 0.000,C 90.000,E1 282.187} C_DIS
LIN {X -0.220,Y -659.414,Z 1002.365,A 0.000,B 0.000,C 90.000,E1 281.715} C_DIS
LIN {X 0.114,Y -658.989,Z 1002.361,A 0.000,B 0.000,C 90.000,E1 280.950} C_DIS
LIN {X -0.222,Y -658.419,Z 1002.358,A 0.000,B 0.000,C 90.000,E1 280.489} C_DIS
LIN {X 0.206,Y -657.573,Z 1002.355,A 0.000,B 0.000,C 90.000,E1 279.962} C_DIS
LIN {X -0.132,Y -656.499,Z 1002.353,A 0.000,B 0.000,C 90.000,E1 279.500} C_DIS
LIN {X 0.278,Y -655.080,Z 1002.350,A 0.000,B 0.000,C 90.000,E1 278.973} C_DIS
LIN {X -0.073,Y -653.295,Z 1002.347,A 0.000,B 0.000,C 90.000,E1 278.511} C_DIS
LIN {X -0.203,Y -652.308,Z 1002.346,A 0.000,B 0.000,C 90.000,E1 278.276} C_DIS
LIN {X 0.077,Y -649.980,Z 1002.343,A 0.000,B 0.000,C 90.000,E1 277.757} C_DIS
LIN {X 0.221,Y -646.258,Z 1002.340,A 0.000,B 0.000,C 90.000,E1 277.125} C_DIS
LIN {X -0.181,Y -642.646,Z 1002.337,A 0.000,B 0.000,C 90.000,E1 276.663} C_DIS
LIN {X -0.091,Y -637.404,Z 1002.333,A 0.000,B 0.000,C 90.000,E1 276.030} C_DIS
LIN {X 0.088,Y -632.694,Z 1002.331,A 0.000,B 0.000,C 90.000,E1 275.511} C_DIS
LIN {X -0.223,Y -627.574,Z 1002.328,A 0.000,B 0.000,C 90.000,E1 275.049} C_DIS
LIN {X 0.275,Y -619.309,Z 1002.324,A 0.000,B 0.000,C 90.000,E1 274.302} C_DIS
LIN {X 0.052,Y -611.794,Z 1002.321,A 0.000,B 0.000,C 90.000,E1 273.784} C_DIS
LIN {X 0.135,Y -605.550,Z 1002.319,A 0.000,B 0.000,C 90.000,E1 273.383} C_DIS
LIN {X -0.066,Y -599.061,Z 1002.317,A 0.000,B 0.000,C 90.000,E1 273.037} C_DIS
LIN {X 0.080,Y -592.123,Z 1002.315,A 0.000,B 0.000,C 90.000,E1 272.694} C_DIS
LIN {X 0.231,Y -584.764,Z 1002.314,A 0.000,B 0.000,C 90.000,E1 272.407} C_DIS
LIN {X -0.264,Y -577.290,Z 1002.312,A 0.000,B 0.000,C 90.000,E1 272.236} C_DIS
LIN {X 0.080,Y -571.559,Z 1002.312,A 0.000,B 0.000,C 90.000,E1 272.064} C_DIS
LIN {X 0.036,Y -564.816,Z 1002.311,A 0.000,B 0.000,C 90.000,E1 271.949} C_DIS
LIN {X 0.060,Y -557.955,Z 1002.311,A 0.000,B 0.000,C 90.000,E1 271.892} C_DIS
LIN {X 0.015,Y -543.562,Z 1002.311,A 0.000,B 0.000,C 90.000,E1 271.892} C_DIS
LIN {X -0.022,Y -542.776,Z 1002.309,A 0.000,B 0.000,C 90.000,E1 271.604} C_DIS
LIN {X 0.092,Y -541.763,Z 1002.303,A 0.000,B 0.000,C 90.000,E1 270.458} C_DIS
LIN {X 0.240,Y -540.611,Z 1002.293,A 0.000,B 0.000,C 90.000,E1 268.740} C_DIS
LIN {X -0.203,Y -539.858,Z 1002.287,A 0.000,B 0.000,C 90.000,E1 267.650} C_DIS
LIN {X -0.055,Y -538.617,Z 1002.277,A 0.000,B 0.000,C 90.000,E1 265.927} C_DIS
LIN {X 0.011,Y -537.694,Z 1002.271,A 0.000,B 0.000,C 90.000,E1 264.780} C_DIS
LIN {X 0.147,Y -536.239,Z 1002.262,A 0.000,B 0.000,C 90.000,E1 263.053} C_DIS
LIN {X -0.193,Y -534.881,Z 1002.254,A 0.000,B 0.000,C 90.000,E1 261.659} C_DIS
LIN {X -0.018,Y -533.411,Z 1002.246,A 0.000,B 0.000,C 90.000,E1 260.208} C_DIS
LIN {X 0.206,Y -531.274,Z 1002.234,A 0.000,B 0.000,C 90.000,E1 258.173} C_DIS
LIN {X -0.001,Y -529.719,Z 1002.227,A 0.000,B 0.000,C 90.000,E1 256.756} C_DIS
LIN {X 0.124,Y -528.473,Z 1002.220,A 0.000,B 0.000,C 90.000,E1 255.589} C_DIS
LIN {X -0.154,Y -525.553,Z 1002.206,A 0.000,B 0.000,C 90.000,E1 253.015} C_DIS
LIN {X 0.177,Y -524.280,Z 1002.199,A 0.000,B 0.000,C 90.000,E1 251.819} C_DIS
LIN {X -0.018,Y -522.860,Z 1002.193,A 0.000,B 0.000,C 90.000,E1 250.678} C_DIS
LIN {X 0.242,Y -520.632,Z 1002.183,A 0.000,B 0.000,C 90.000,E1 248.901} C_DIS
LIN {X -0.174,Y -518.727,Z 1002.175,A 0.000,B 0.000,C 90.000,E1 247.486} C_DIS
LIN {X -0.227,Y -517.609,Z 1002.170,A 0.000,B 0.000,C 90.000,E1 246.613} C_DIS
LIN {X 0.183,Y -515.393,Z 1002.162,A 0.000,B 0.000,C 90.000,E1 245.101} C_DIS
LIN {X 0.088,Y -514.109,Z 1002.157,A 0.000,B 0.000,C 90.000,E1 244.229} C_DIS
LIN {X -0.162,Y -511.261,Z 1002.147,A 0.000,B 0.000,C 90.000,E1 242.487} C_DIS
LIN {X -0.110,Y -508.913,Z 1002.139,A 0.000,B 0.000,C 90.000,E1 241.001} C_DIS
LIN {X -0.300,Y -506.314,Z 1002.131,A 0.000,B 0.000,C 90.000,E1 239.537} C_DIS
LIN {X -0.153,Y -504.100,Z 1002.124,A 0.000,B 0.000,C 90.000,E1 238.329} C_DIS
LIN {X 0.133,Y -500.466,Z 1002.114,A 0.000,B 0.000,C 90.000,E1 236.501} C_DIS
LIN {X -0.083,Y -497.124,Z 1002.106,A 0.000,B 0.000,C 90.000,E1 235.022} C_DIS
LIN {X 0.185,Y -494.295,Z 1002.099,A 0.000,B 0.000,C 90.000,E1 233.783} C_DIS
LIN {X -0.021,Y -488.310,Z 1002.085,A 0.000,B 0.000,C 90.000,E1 231.376} C_DIS
LIN {X -0.002,Y -485.390,Z 1002.079,A 0.000,B 0.000,C 90.000,E1 230.150} C_DIS
LIN {X 0.038,Y -481.868,Z 1002.070,A 0.000,B 0.000,C 90.000,E1 228.609} C_DIS
LIN {X 0.149,Y -475.826,Z 1002.055,A 0.000,B 0.000,C 90.000,E1 225.810} C_DIS
LIN {X -0.002,Y -472.598,Z 1002.046,A 0.000,B 0.000,C 90.000,E1 224.271} C_DIS
LIN {X 0.124,Y -469.293,Z 1002.037,A 0.000,B 0.000,C 90.000,E1 222.690} C_DIS
LIN {X 0.038,Y -464.490,Z 1002.025,A 0.000,B 0.000,C 90.000,E1 220.496} C_DIS
LIN {X 0.075,Y -460.130,Z 1002.014,A 0.000,B 0.000,C 90.000,E1 218.588} C_DIS
LIN {X -0.117,Y -455.270,Z 1002.002,A 0.000,B 0.000,C 90.000,E1 216.377} C_DIS
LIN {X 0.133,Y -451.764,Z 1001.993,A 0.000,B 0.000,C 90.000,E1 214.739} C_DIS
LIN {X -0.123,Y -447.561,Z 1001.982,A 0.000,B 0.000,C 90.000,E1 212.832} C_DIS
LIN {X -0.088,Y -443.327,Z 1001.971,A 0.000,B 0.000,C 90.000,E1 210.875} C_DIS
LIN {X 0.173,Y -439.688,Z 1001.962,A 0.000,B 0.000,C 90.000,E1 209.205} C_DIS
LIN {X -0.068,Y -435.929,Z 1001.953,A 0.000,B 0.000,C 90.000,E1 207.590} C_DIS
LIN {X 0.014,Y -432.248,Z 1001.944,A 0.000,B 0.000,C 90.000,E1 205.924} C_DIS
LIN {X 0.028,Y -429.179,Z 1001.937,A 0.000,B 0.000,C 90.000,E1 204.591} C_DIS
LIN {X -0.070,Y -423.972,Z 1001.924,A 0.000,B 0.000,C 90.000,E1 202.259} C_DIS
LIN {X -0.231,Y -418.225,Z 1001.909,A 0.000,B 0.000,C 90.000,E1 199.577} C_DIS
LIN {X -0.003,Y -411.236,Z 1001.888,A 0.000,B 0.000,C 90.000,E1 195.788} C_DIS
LIN {X 0.150,Y -406.660,Z 1001.872,A 0.000,B 0.000,C 90.000,E1 193.008} C_DIS
LIN {X -0.032,Y -403.959,Z 1001.863,A 0.000,B 0.000,C 90.000,E1 191.299} C_DIS
LIN {X -0.038,Y -400.804,Z 1001.851,A 0.000,B 0.000,C 90.000,E1 189.208} C_DIS
LIN {X -0.057,Y -400.038,Z 1001.847,A 0.000,B 0.000,C 90.000,E1 188.511} C_DIS
LIN {X -0.099,Y -399.332,Z 1001.841,A 0.000,B 0.000,C 90.000,E1 187.466} C_DIS
LIN {X -0.184,Y -399.521,Z 1001.838,A 0.000,B 0.000,C 90.000,E1 186.777} C_DIS
LIN {X 0.131,Y -400.253,Z 1001.834,A 0.000,B 0.000,C 90.000,E1 186.030} C_DIS
LIN {X -0.184,Y -401.897,Z 1001.830,A 0.000,B 0.000,C 90.000,E1 185.391} C_DIS
LIN {X 0.164,Y -403.172,Z 1001.828,A 0.000,B 0.000,C 90.000,E1 184.992} C_DIS
LIN {X -0.072,Y -404.526,Z 1001.826,A 0.000,B 0.000,C 90.000,E1 184.702} C_DIS
LIN {X -0.131,Y -407.324,Z 1001.823,A 0.000,B 0.000,C 90.000,E1 184.188} C_DIS
LIN {X -0.143,Y -410.977,Z 1001.820,A 0.000,B 0.000,C 90.000,E1 183.669} C_DIS
LIN {X -0.013,Y -417.896,Z 1001.816,A 0.000,B 0.000,C 90.000,E1 182.808} C_DIS
LIN {X -0.057,Y -429.347,Z 1001.809,A 0.000,B 0.000,C 90.000,E1 181.547} C_DIS
LIN {X -0.072,Y -443.464,Z 1001.800,A 0.000,B 0.000,C 90.000,E1 180.000} C_DIS
LIN {X -0.039,Y -454.356,Z 1001.793,A 0.000,B 0.000,C 90.000,E1 178.797} C_DIS
LIN {X -0.044,Y -462.505,Z 1001.788,A 0.000,B 0.000,C 90.000,E1 177.879} C_DIS
LIN {X 0.190,Y -469.083,Z 1001.784,A 0.000,B 0.000,C 90.000,E1 177.078} C_DIS
LIN {X 0.024,Y -476.787,Z 1001.779,A 0.000,B 0.000,C 90.000,E1 176.159} C_DIS
LIN {X -0.224,Y -482.932,Z 1001.774,A 0.000,B 0.000,C 90.000,E1 175.412} C_DIS
LIN {X -0.221,Y -489.665,Z 1001.769,A 0.000,B 0.000,C 90.000,E1 174.489} C_DIS
LIN {X 0.033,Y -497.138,Z 1001.763,A 0.000,B 0.000,C 90.000,E1 173.394} C_DIS
LIN {X -0.109,Y -504.312,Z 1001.758,A 0.000,B 0.000,C 90.000,E1 172.356} C_DIS
LIN {X -0.092,Y -511.319,Z 1001.752,A 0.000,B 0.000,C 90.000,E1 171.310} C_DIS
LIN {X 0.218,Y -520.641,Z 1001.744,A 0.000,B 0.000,C 90.000,E1 169.803} C_DIS
LIN {X 0.281,Y -529.450,Z 1001.735,A 0.000,B 0.000,C 90.000,E1 168.342} C_DIS
LIN {X 0.041,Y -539.781,Z 1001.726,A 0.000,B 0.000,C 90.000,E1 166.645} C_DIS
LIN {X -0.111,Y -548.735,Z 1001.717,A 0.000,B 0.000,C 90.000,E1 165.102} C_DIS
LIN {X 0.059,Y -554.318,Z 1001.712,A 0.000,B 0.000,C 90.000,E1 164.102} C_DIS
LIN {X 0.044,Y -561.083,Z 1001.705,A 0.000,B 0.000,C 90.000,E1 162.851} C_DIS
LIN {X 0.201,Y -568.415,Z 1001.697,A 0.000,B 0.000,C 90.000,E1 161.456} C_DIS
LIN {X -0.314,Y -573.217,Z 1001.692,A 0.000,B 0.000,C 90.000,E1 160.550} C_DIS
LIN {X -0.039,Y -577.865,Z 1001.687,A 0.000,B 0.000,C 90.000,E1 159.571} C_DIS
LIN {X 0.225,Y -582.928,Z 1001.681,A 0.000,B 0.000,C 90.000,E1 158.465} C_DIS
LIN {X 0.208,Y -585.920,Z 1001.677,A 0.000,B 0.000,C 90.000,E1 157.794} C_DIS
LIN {X 0.149,Y -589.449,Z 1001.672,A 0.000,B 0.000,C 90.000,E1 156.997} C_DIS
LIN {X 0.251,Y -593.739,Z 1001.666,A 0.000,B 0.000,C 90.000,E1 155.921} C_DIS
LIN {X -0.119,Y -597.626,Z 1001.661,A 0.000,B 0.000,C 90.000,E1 154.897} C_DIS
LIN {X -0.079,Y -600.371,Z 1001.656,A 0.000,B 0.000,C 90.000,E1 154.101} C_DIS
LIN {X -0.092,Y -603.599,Z 1001.650,A 0.000,B 0.000,C 90.000,E1 153.050} C_DIS
LIN {X 0.099,Y -608.247,Z 1001.642,A 0.000,B 0.000,C 90.000,E1 151.463} C_DIS
LIN {X -0.105,Y -612.657,Z 1001.633,A 0.000,B 0.000,C 90.000,E1 149.921} C_DIS
LIN {X 0.066,Y -615.544,Z 1001.627,A 0.000,B 0.000,C 90.000,E1 148.869} C_DIS
LIN {X 0.043,Y -619.042,Z 1001.620,A 0.000,B 0.000,C 90.000,E1 147.582} C_DIS
LIN {X 0.198,Y -624.588,Z 1001.609,A 0.000,B 0.000,C 90.000,E1 145.515} C_DIS
LIN {X 0.150,Y -628.802,Z 1001.600,A 0.000,B 0.000,C 90.000,E1 143.989} C_DIS
LIN {X 0.042,Y -632.884,Z 1001.592,A 0.000,B 0.000,C 90.000,E1 142.477} C_DIS
LIN {X 0.148,Y -635.629,Z 1001.586,A 0.000,B 0.000,C 90.000,E1 141.457} C_DIS
LIN {X 0.184,Y -638.975,Z 1001.579,A 0.000,B 0.000,C 90.000,E1 140.194} C_DIS
LIN {X 0.272,Y -642.256,Z 1001.572,A 0.000,B 0.000,C 90.000,E1 138.933} C_DIS
LIN {X 0.185,Y -647.482,Z 1001.561,A 0.000,B 0.000,C 90.000,E1 136.944} C_DIS
LIN {X -0.216,Y -652.356,Z 1001.551,A 0.000,B 0.000,C 90.000,E1 135.243} C_DIS
LIN {X 0.006,Y -656.912,Z 1001.543,A 0.000,B 0.000,C 90.000,E1 133.743} C_DIS
LIN {X 0.289,Y -663.376,Z 1001.532,A 0.000,B 0.000,C 90.000,E1 131.757} C_DIS
LIN {X 0.287,Y -667.507,Z 1001.525,A 0.000,B 0.000,C 90.000,E1 130.539} C_DIS
LIN {X -0.081,Y -672.191,Z 1001.517,A 0.000,B 0.000,C 90.000,E1 129.116} C_DIS
LIN {X 0.151,Y -675.739,Z 1001.511,A 0.000,B 0.000,C 90.000,E1 127.890} C_DIS
LIN {X 0.053,Y -679.906,Z 1001.503,A 0.000,B 0.000,C 90.000,E1 126.457} C_DIS
LIN {X 0.017,Y -683.230,Z 1001.496,A 0.000,B 0.000,C 90.000,E1 125.264} C_DIS
LIN {X 0.034,Y -686.506,Z 1001.489,A 0.000,B 0.000,C 90.000,E1 124.072} C_DIS
LIN {X 0.082,Y -688.970,Z 1001.484,A 0.000,B 0.000,C 90.000,E1 123.118} C_DIS
LIN {X -0.190,Y -692.578,Z 1001.476,A 0.000,B 0.000,C 90.000,E1 121.720} C_DIS
LIN {X -0.191,Y -695.510,Z 1001.470,A 0.000,B 0.000,C 90.000,E1 120.541} C_DIS
LIN {X -0.046,Y -697.535,Z 1001.464,A 0.000,B 0.000,C 90.000,E1 119.589} C_DIS
LIN {X 0.382,Y -699.078,Z 1001.459,A 0.000,B 0.000,C 90.000,E1 118.615} C_DIS
LIN {X -0.381,Y -700.015,Z 1001.455,A 0.000,B 0.000,C 90.000,E1 117.975} C_DIS
LIN {X 0.162,Y -700.453,Z 1001.453,A 0.000,B 0.000,C 90.000,E1 117.462} C_DIS
LIN {X -0.109,Y -701.784,Z 1001.444,A 0.000,B 0.000,C 90.000,E1 115.848} C_DIS
LIN {X 0.066,Y -702.456,Z 1001.438,A 0.000,B 0.000,C 90.000,E1 114.899} C_DIS
LIN {X -0.030,Y -702.620,Z 1001.435,A 0.000,B 0.000,C 90.000,E1 114.207} C_DIS
LIN {X -0.402,Y -702.088,Z 1001.432,A 0.000,B 0.000,C 90.000,E1 113.770} C_DIS
LIN {X -0.127,Y -701.708,Z 1001.431,A 0.000,B 0.000,C 90.000,E1 113.515} C_DIS
LIN {X 0.277,Y -699.093,Z 1001.427,A 0.000,B 0.000,C 90.000,E1 112.898} C_DIS
LIN {X -0.234,Y -698.363,Z 1001.427,A 0.000,B 0.000,C 90.000,E1 112.823} C_DIS
LIN {X -0.104,Y -697.271,Z 1001.426,A 0.000,B 0.000,C 90.000,E1 112.695} C_DIS
LIN {X -0.256,Y -691.635,Z 1001.424,A 0.000,B 0.000,C 90.000,E1 112.280} C_DIS
LIN {X 0.053,Y -689.899,Z 1001.423,A 0.000,B 0.000,C 90.000,E1 112.153} C_DIS
LIN {X 0.098,Y -684.870,Z 1001.422,A 0.000,B 0.000,C 90.000,E1 111.972} C_DIS
LIN {X -0.051,Y -679.925,Z 1001.422,A 0.000,B 0.000,C 90.000,E1 111.897} C_DIS
LIN {X -0.159,Y -675.720,Z 1001.421,A 0.000,B 0.000,C 90.000,E1 111.844} C_DIS
LIN {X -0.261,Y -672.150,Z 1001.421,A 0.000,B 0.000,C 90.000,E1 111.844} C_DIS
LIN {X -0.274,Y -618.747,Z 1001.421,A 0.000,B 0.000,C 90.000,E1 111.844} C_DIS
LIN {X -0.215,Y -615.495,Z 1001.421,A 0.000,B 0.000,C 90.000,E1 111.770} C_DIS
LIN {X 0.075,Y -610.005,Z 1001.420,A 0.000,B 0.000,C 90.000,E1 111.589} C_DIS
LIN {X -0.085,Y -602.096,Z 1001.418,A 0.000,B 0.000,C 90.000,E1 111.280} C_DIS
LIN {X -0.162,Y -599.409,Z 1001.417,A 0.000,B 0.000,C 90.000,E1 111.153} C_DIS
LIN {X 0.052,Y -594.703,Z 1001.416,A 0.000,B 0.000,C 90.000,E1 110.865} C_DIS
LIN {X 0.003,Y -587.929,Z 1001.413,A 0.000,B 0.000,C 90.000,E1 110.375} C_DIS
LIN {X -0.050,Y -578.055,Z 1001.409,A 0.000,B 0.000,C 90.000,E1 109.577} C_DIS
LIN {X -0.227,Y -572.196,Z 1001.406,A 0.000,B 0.000,C 90.000,E1 109.141} C_DIS
LIN {X 0.315,Y -563.791,Z 1001.404,A 0.000,B 0.000,C 90.000,E1 108.598} C_DIS
LIN {X 0.169,Y -550.525,Z 1001.400,A 0.000,B 0.000,C 90.000,E1 107.946} C_DIS
LIN {X -0.254,Y -548.985,Z 1001.399,A 0.000,B 0.000,C 90.000,E1 107.819} C_DIS
LIN {X 0.227,Y -548.961,Z 1001.399,A 0.000,B 0.000,C 90.000,E1 107.764} C_DIS
LIN {X 0.088,Y -548.559,Z 1001.397,A 0.000,B 0.000,C 90.000,E1 107.511} C_DIS
LIN {X -0.094,Y -548.477,Z 1001.394,A 0.000,B 0.000,C 90.000,E1 106.968} C_DIS
LIN {X -0.091,Y -548.991,Z 1001.388,A 0.000,B 0.000,C 90.000,E1 105.843} C_DIS
LIN {X -0.156,Y -549.952,Z 1001.377,A 0.000,B 0.000,C 90.000,E1 103.883} C_DIS
LIN {X 0.254,Y -552.949,Z 1001.357,A 0.000,B 0.000,C 90.000,E1 100.197} C_DIS
LIN {X -0.074,Y -555.083,Z 1001.346,A 0.000,B 0.000,C 90.000,E1 98.276} C_DIS
LIN {X -0.151,Y -556.567,Z 1001.338,A 0.000,B 0.000,C 90.000,E1 96.891} C_DIS
LIN {X -0.258,Y -557.853,Z 1001.331,A 0.000,B 0.000,C 90.000,E1 95.511} C_DIS
LIN {X 0.141,Y -558.679,Z 1001.324,A 0.000,B 0.000,C 90.000,E1 94.359} C_DIS
LIN {X 0.069,Y -559.536,Z 1001.317,A 0.000,B 0.000,C 90.000,E1 92.980} C_DIS
LIN {X -0.024,Y -560.169,Z 1001.309,A 0.000,B 0.000,C 90.000,E1 91.604} C_DIS
LIN {X -0.117,Y -560.941,Z 1001.301,A 0.000,B 0.000,C 90.000,E1 90.229} C_DIS
LIN {X -0.002,Y -561.735,Z 1001.291,A 0.000,B 0.000,C 90.000,E1 88.282} C_DIS
LIN {X -0.059,Y -561.990,Z 1001.283,A 0.000,B 0.000,C 90.000,E1 86.906} C_DIS
LIN {X -0.076,Y -562.193,Z 1001.275,A 0.000,B 0.000,C 90.000,E1 85.527} C_DIS
LIN {X -0.086,Y -562.405,Z 1001.267,A 0.000,B 0.000,C 90.000,E1 84.147} C_DIS
LIN {X 0.196,Y -562.742,Z 1001.257,A 0.000,B 0.000,C 90.000,E1 82.186} C_DIS
LIN {X 0.002,Y -563.255,Z 1001.246,A 0.000,B 0.000,C 90.000,E1 80.274} C_DIS
LIN {X 0.028,Y -564.080,Z 1001.235,A 0.000,B 0.000,C 90.000,E1 78.342} C_DIS
LIN {X 0.302,Y -564.811,Z 1001.228,A 0.000,B 0.000,C 90.000,E1 76.937} C_DIS
LIN {X -0.049,Y -565.964,Z 1001.217,A 0.000,B 0.000,C 90.000,E1 75.046} C_DIS
LIN {X -0.168,Y -566.966,Z 1001.209,A 0.000,B 0.000,C 90.000,E1 73.685} C_DIS
LIN {X -0.165,Y -568.458,Z 1001.199,A 0.000,B 0.000,C 90.000,E1 71.764} C_DIS
LIN {X -0.101,Y -569.584,Z 1001.190,A 0.000,B 0.000,C 90.000,E1 70.115} C_DIS
LIN {X 0.347,Y -570.727,Z 1001.179,A 0.000,B 0.000,C 90.000,E1 68.156} C_DIS
LIN {X -0.254,Y -571.656,Z 1001.168,A 0.000,B 0.000,C 90.000,E1 66.305} C_DIS
LIN {X -0.214,Y -572.342,Z 1001.159,A 0.000,B 0.000,C 90.000,E1 64.665} C_DIS
LIN {X 0.250,Y -572.784,Z 1001.152,A 0.000,B 0.000,C 90.000,E1 63.256} C_DIS
LIN {X 0.055,Y -573.276,Z 1001.143,A 0.000,B 0.000,C 90.000,E1 61.641} C_DIS
LIN {X 0.143,Y -573.717,Z 1001.133,A 0.000,B 0.000,C 90.000,E1 59.999} C_DIS
LIN {X -0.096,Y -574.009,Z 1001.126,A 0.000,B 0.000,C 90.000,E1 58.663} C_DIS
LIN {X -0.194,Y -574.216,Z 1001.117,A 0.000,B 0.000,C 90.000,E1 57.041} C_DIS
LIN {X -0.122,Y -574.435,Z 1001.109,A 0.000,B 0.000,C 90.000,E1 55.674} C_DIS
LIN {X -0.017,Y -574.463,Z 1001.105,A 0.000,B 0.000,C 90.000,E1 54.848} C_DIS
LIN {X -0.091,Y -574.337,Z 1001.097,A 0.000,B 0.000,C 90.000,E1 53.497} C_DIS
LIN {X -0.110,Y -574.140,Z 1001.093,A 0.000,B 0.000,C 90.000,E1 52.683} C_DIS
LIN {X -0.334,Y -573.601,Z 1001.087,A 0.000,B 0.000,C 90.000,E1 51.618} C_DIS
LIN {X -0.076,Y -572.821,Z 1001.079,A 0.000,B 0.000,C 90.000,E1 50.231} C_DIS
LIN {X 0.093,Y -571.707,Z 1001.071,A 0.000,B 0.000,C 90.000,E1 48.852} C_DIS
LIN {X 0.127,Y -570.658,Z 1001.065,A 0.000,B 0.000,C 90.000,E1 47.757} C_DIS
LIN {X 0.062,Y -569.677,Z 1001.061,A 0.000,B 0.000,C 90.000,E1 46.944} C_DIS
LIN {X -0.349,Y -567.962,Z 1001.055,A 0.000,B 0.000,C 90.000,E1 45.891} C_DIS
LIN {X -0.066,Y -566.471,Z 1001.050,A 0.000,B 0.000,C 90.000,E1 45.040} C_DIS
LIN {X -0.114,Y -564.265,Z 1001.044,A 0.000,B 0.000,C 90.000,E1 43.947} C_DIS
LIN {X 0.135,Y -562.381,Z 1001.040,A 0.000,B 0.000,C 90.000,E1 43.095} C_DIS
LIN {X -0.048,Y -560.141,Z 1001.035,A 0.000,B 0.000,C 90.000,E1 42.285} C_DIS
LIN {X 0.154,Y -557.672,Z 1001.030,A 0.000,B 0.000,C 90.000,E1 41.434} C_DIS
LIN {X -0.111,Y -555.867,Z 1001.027,A 0.000,B 0.000,C 90.000,E1 40.906} C_DIS
LIN {X 0.037,Y -553.940,Z 1001.024,A 0.000,B 0.000,C 90.000,E1 40.334} C_DIS
LIN {X 0.105,Y -551.861,Z 1001.021,A 0.000,B 0.000,C 90.000,E1 39.769} C_DIS
LIN {X -0.144,Y -548.367,Z 1001.016,A 0.000,B 0.000,C 90.000,E1 38.955} C_DIS
LIN {X -0.150,Y -543.941,Z 1001.011,A 0.000,B 0.000,C 90.000,E1 37.971} C_DIS
LIN {X 0.274,Y -539.821,Z 1001.006,A 0.000,B 0.000,C 90.000,E1 37.076} C_DIS
LIN {X 0.164,Y -534.738,Z 1001.001,A 0.000,B 0.000,C 90.000,E1 36.091} C_DIS
LIN {X 0.154,Y -530.036,Z 1000.996,A 0.000,B 0.000,C 90.000,E1 35.231} C_DIS
LIN {X -0.025,Y -527.590,Z 1000.993,A 0.000,B 0.000,C 90.000,E1 34.818} C_DIS
LIN {X 0.314,Y -522.402,Z 1000.989,A 0.000,B 0.000,C 90.000,E1 33.913} C_DIS
LIN {X -0.130,Y -516.849,Z 1000.984,A 0.000,B 0.000,C 90.000,E1 33.086} C_DIS
LIN {X 0.161,Y -512.850,Z 1000.981,A 0.000,B 0.000,C 90.000,E1 32.467} C_DIS
LIN {X 0.147,Y -508.639,Z 1000.977,A 0.000,B 0.000,C 90.000,E1 31.878} C_DIS
LIN {X -0.104,Y -505.379,Z 1000.975,A 0.000,B 0.000,C 90.000,E1 31.465} C_DIS
LIN {X -0.044,Y -500.754,Z 1000.972,A 0.000,B 0.000,C 90.000,E1 30.875} C_DIS
LIN {X 0.060,Y -496.978,Z 1000.969,A 0.000,B 0.000,C 90.000,E1 30.413} C_DIS
LIN {X -0.013,Y -488.867,Z 1000.964,A 0.000,B 0.000,C 90.000,E1 29.539} C_DIS
LIN {X 0.092,Y -483.310,Z 1000.961,A 0.000,B 0.000,C 90.000,E1 28.949} C_DIS
LIN {X 0.165,Y -474.666,Z 1000.956,A 0.000,B 0.000,C 90.000,E1 28.103} C_DIS
LIN {X -0.059,Y -465.989,Z 1000.952,A 0.000,B 0.000,C 90.000,E1 27.308} C_DIS
LIN {X 0.064,Y -456.984,Z 1000.947,A 0.000,B 0.000,C 90.000,E1 26.488} C_DIS
LIN {X 0.016,Y -446.413,Z 1000.942,A 0.000,B 0.000,C 90.000,E1 25.591} C_DIS
LIN {X 0.031,Y -425.732,Z 1000.932,A 0.000,B 0.000,C 90.000,E1 23.770} C_DIS
LIN {X 0.154,Y -412.455,Z 1000.925,A 0.000,B 0.000,C 90.000,E1 22.461} C_DIS
LIN {X -0.063,Y -399.606,Z 1000.917,A 0.000,B 0.000,C 90.000,E1 21.099} C_DIS
LIN {X 0.046,Y -397.225,Z 1000.916,A 0.000,B 0.000,C 90.000,E1 20.791} C_DIS
LIN {X 0.101,Y -394.458,Z 1000.913,A 0.000,B 0.000,C 90.000,E1 20.375} C_DIS
LIN {X -0.087,Y -393.626,Z 1000.912,A 0.000,B 0.000,C 90.000,E1 20.248} C_DIS
LIN {X -0.011,Y -391.394,Z 1000.909,A 0.000,B 0.000,C 90.000,E1 19.704} C_DIS
LIN {X 0.209,Y -390.422,Z 1000.907,A 0.000,B 0.000,C 90.000,E1 19.141} C_DIS
LIN {X 0.039,Y -390.370,Z 1000.903,A 0.000,B 0.000,C 90.000,E1 18.544} C_DIS
LIN {X 0.212,Y -391.494,Z 1000.895,A 0.000,B 0.000,C 90.000,E1 17.094} C_DIS
LIN {X -0.049,Y -394.034,Z 1000.881,A 0.000,B 0.000,C 90.000,E1 14.647} C_DIS
LIN {X -0.160,Y -399.199,Z 1000.860,A 0.000,B 0.000,C 90.000,E1 10.782} C_DIS
LIN {X 0.119,Y -406.488,Z 1000.837,A 0.000,B 0.000,C 90.000,E1 6.549} C_DIS
LIN {X 0.121,Y -412.298,Z 1000.821,A 0.000,B 0.000,C 90.000,E1 3.784} C_DIS
LIN {X 0.192,Y -417.340,Z 1000.809,A 0.000,B 0.000,C 90.000,E1 1.547} C_DIS
LIN {X 0.155,Y -419.436,Z 1000.806,A 0.000,B 0.000,C 90.000,E1 0.974} C_DIS
LIN {X 0.127,Y -422.393,Z 1000.803,A 0.000,B 0.000,C 90.000,E1 0.458} C_DIS
LIN {X 0.145,Y -423.440,Z 1000.802,A 0.000,B 0.000,C 90.000,E1 0.286} C_DIS
LIN {X 0.080,Y -427.751,Z 1000.799,A 0.000,B 0.000,C 90.000,E1 359.885} C_DIS
LIN {X 0.162,Y -429.082,Z 1000.799,A 0.000,B 0.000,C 90.000,E1 359.771} C_DIS
LIN {X -0.199,Y -434.497,Z 1000.797,A 0.000,B 0.000,C 90.000,E1 359.484} C_DIS
LIN {X 0.174,Y -440.906,Z 1000.795,A 0.000,B 0.000,C 90.000,E1 359.083} C_DIS
LIN {X 0.130,Y -454.113,Z 1000.791,A 0.000,B 0.000,C 90.000,E1 358.339} C_DIS
LIN {X 0.100,Y -469.020,Z 1000.786,A 0.000,B 0.000,C 90.000,E1 357.478} C_DIS
LIN {X -0.003,Y -482.310,Z 1000.782,A 0.000,B 0.000,C 90.000,E1 356.731} C_DIS
LIN {X -0.129,Y -490.602,Z 1000.779,A 0.000,B 0.000,C 90.000,E1 356.274} C_DIS
LIN {X -0.171,Y -503.162,Z 1000.775,A 0.000,B 0.000,C 90.000,E1 355.527} C_DIS
LIN {X 0.229,Y -512.390,Z 1000.772,A 0.000,B 0.000,C 90.000,E1 354.894} C_DIS
LIN {X 0.088,Y -519.997,Z 1000.769,A 0.000,B 0.000,C 90.000,E1 354.375} C_DIS
LIN {X 0.219,Y -527.531,Z 1000.766,A 0.000,B 0.000,C 90.000,E1 353.799} C_DIS
LIN {X -0.204,Y -535.902,Z 1000.762,A 0.000,B 0.000,C 90.000,E1 353.166} C_DIS
LIN {X -0.079,Y -542.674,Z 1000.759,A 0.000,B 0.000,C 90.000,E1 352.534} C_DIS
LIN {X 0.250,Y -549.189,Z 1000.755,A 0.000,B 0.000,C 90.000,E1 351.837} C_DIS
LIN {X 0.008,Y -554.276,Z 1000.752,A 0.000,B 0.000,C 90.000,E1 351.319} C_DIS
LIN {X 0.014,Y -560.001,Z 1000.748,A 0.000,B 0.000,C 90.000,E1 350.622} C_DIS
LIN {X 0.001,Y -563.282,Z 1000.746,A 0.000,B 0.000,C 90.000,E1 350.208} C_DIS
LIN {X 0.083,Y -568.041,Z 1000.742,A 0.000,B 0.000,C 90.000,E1 349.511} C_DIS
LIN {X 0.205,Y -572.302,Z 1000.738,A 0.000,B 0.000,C 90.000,E1 348.814} C_DIS
LIN {X -0.203,Y -576.229,Z 1000.734,A 0.000,B 0.000,C 90.000,E1 348.173} C_DIS
LIN {X -0.239,Y -581.379,Z 1000.729,A 0.000,B 0.000,C 90.000,E1 347.229} C_DIS
LIN {X 0.041,Y -587.434,Z 1000.722,A 0.000,B 0.000,C 90.000,E1 345.992} C_DIS
LIN {X -0.159,Y -593.120,Z 1000.716,A 0.000,B 0.000,C 90.000,E1 344.810} C_DIS
LIN {X -0.053,Y -597.861,Z 1000.710,A 0.000,B 0.000,C 90.000,E1 343.740} C_DIS
LIN {X 0.106,Y -602.338,Z 1000.704,A 0.000,B 0.000,C 90.000,E1 342.670} C_DIS
LIN {X -0.343,Y -607.551,Z 1000.697,A 0.000,B 0.000,C 90.000,E1 341.402} C_DIS
LIN {X 0.072,Y -612.505,Z 1000.689,A 0.000,B 0.000,C 90.000,E1 340.061} C_DIS
LIN {X 0.036,Y -615.925,Z 1000.684,A 0.000,B 0.000,C 90.000,E1 339.028} C_DIS
LIN {X 0.268,Y -619.076,Z 1000.678,A 0.000,B 0.000,C 90.000,E1 337.975} C_DIS
LIN {X -0.025,Y -622.177,Z 1000.672,A 0.000,B 0.000,C 90.000,E1 336.975} C_DIS
LIN {X 0.296,Y -625.050,Z 1000.666,A 0.000,B 0.000,C 90.000,E1 335.921} C_DIS
LIN {X 0.094,Y -628.267,Z 1000.659,A 0.000,B 0.000,C 90.000,E1 334.665} C_DIS
LIN {X 0.185,Y -630.682,Z 1000.654,A 0.000,B 0.000,C 90.000,E1 333.640} C_DIS
LIN {X 0.277,Y -632.300,Z 1000.649,A 0.000,B 0.000,C 90.000,E1 332.871} C_DIS
LIN {X -0.058,Y -635.265,Z 1000.641,A 0.000,B 0.000,C 90.000,E1 331.385} C_DIS
LIN {X -0.034,Y -637.899,Z 1000.633,A 0.000,B 0.000,C 90.000,E1 329.871} C_DIS
LIN {X -0.017,Y -639.867,Z 1000.626,A 0.000,B 0.000,C 90.000,E1 328.614} C_DIS
LIN {X -0.077,Y -640.878,Z 1000.622,A 0.000,B 0.000,C 90.000,E1 327.867} C_DIS
LIN {X -0.215,Y -642.380,Z 1000.615,A 0.000,B 0.000,C 90.000,E1 326.628} C_DIS
LIN {X 0.159,Y -643.389,Z 1000.609,A 0.000,B 0.000,C 90.000,E1 325.595} C_DIS
LIN {X 0.016,Y -644.223,Z 1000.603,A 0.000,B 0.000,C 90.000,E1 324.609} C_DIS
LIN {X 0.303,Y -644.912,Z 1000.596,A 0.000,B 0.000,C 90.000,E1 323.336} C_DIS
LIN {X 0.084,Y -645.493,Z 1000.590,A 0.000,B 0.000,C 90.000,E1 322.110} C_DIS
LIN {X -0.212,Y -646.031,Z 1000.581,A 0.000,B 0.000,C 90.000,E1 320.642} C_DIS
LIN {X -0.233,Y -646.946,Z 1000.569,A 0.000,B 0.000,C 90.000,E1 318.405} C_DIS
LIN {X -0.143,Y -647.922,Z 1000.561,A 0.000,B 0.000,C 90.000,E1 316.905} C_DIS
LIN {X -0.085,Y -648.887,Z 1000.551,A 0.000,B 0.000,C 90.000,E1 315.162} C_DIS
LIN {X -0.056,Y -650.293,Z 1000.540,A 0.000,B 0.000,C 90.000,E1 313.176} C_DIS
LIN {X 0.104,Y -651.286,Z 1000.532,A 0.000,B 0.000,C 90.000,E1 311.676} C_DIS
LIN {X 0.333,Y -652.126,Z 1000.523,A 0.000,B 0.000,C 90.000,E1 310.172} C_DIS
LIN {X 0.106,Y -652.876,Z 1000.514,A 0.000,B 0.000,C 90.000,E1 308.463} C_DIS
LIN {X 0.012,Y -653.346,Z 1000.507,A 0.000,B 0.000,C 90.000,E1 307.237} C_DIS
LIN {X -0.067,Y -653.565,Z 1000.503,A 0.000,B 0.000,C 90.000,E1 306.503} C_DIS
LIN {X -0.087,Y -653.790,Z 1000.495,A 0.000,B 0.000,C 90.000,E1 305.025} C_DIS
LIN {X -0.022,Y -654.158,Z 1000.485,A 0.000,B 0.000,C 90.000,E1 303.293} C_DIS
LIN {X -0.113,Y -659.061,Z 1000.454,A 0.000,B 0.000,C 90.000,E1 297.641} C_DIS
LIN {X 0.071,Y -661.122,Z 1000.445,A 0.000,B 0.000,C 90.000,E1 296.155} C_DIS
LIN {X -0.139,Y -662.878,Z 1000.439,A 0.000,B 0.000,C 90.000,E1 294.951} C_DIS
LIN {X 0.002,Y -663.802,Z 1000.435,A 0.000,B 0.000,C 90.000,E1 294.207} C_DIS
LIN {X 0.300,Y -664.854,Z 1000.429,A 0.000,B 0.000,C 90.000,E1 293.206} C_DIS
LIN {X -0.147,Y -665.322,Z 1000.425,A 0.000,B 0.000,C 90.000,E1 292.514} C_DIS
LIN {X -0.118,Y -665.456,Z 1000.422,A 0.000,B 0.000,C 90.000,E1 292.025} C_DIS
LIN {X -0.086,Y -665.100,Z 1000.420,A 0.000,B 0.000,C 90.000,E1 291.535} C_DIS
LIN {X 0.051,Y -664.795,Z 1000.418,A 0.000,B 0.000,C 90.000,E1 291.280} C_DIS
LIN {X 0.080,Y -663.136,Z 1000.416,A 0.000,B 0.000,C 90.000,E1 290.791} C_DIS
LIN {X -0.024,Y -661.912,Z 1000.414,A 0.000,B 0.000,C 90.000,E1 290.556} C_DIS
LIN {X 0.100,Y -660.056,Z 1000.413,A 0.000,B 0.000,C 90.000,E1 290.301} C_DIS
LIN {X 0.104,Y -656.282,Z 1000.411,A 0.000,B 0.000,C 90.000,E1 289.939} C_DIS
LIN {X 0.055,Y -651.302,Z 1000.409,A 0.000,B 0.000,C 90.000,E1 289.631} C_DIS
LIN {X 0.301,Y -648.774,Z 1000.408,A 0.000,B 0.000,C 90.000,E1 289.450} C_DIS
LIN {X -0.061,Y -642.606,Z 1000.406,A 0.000,B 0.000,C 90.000,E1 289.141} C_DIS
LIN {X -0.333,Y -638.392,Z 1000.405,A 0.000,B 0.000,C 90.000,E1 288.906} C_DIS
LIN {X 0.155,Y -638.202,Z 1000.405,A 0.000,B 0.000,C 90.000,E1 288.852} C_DIS
LIN {X 0.097,Y -638.160,Z 1000.405,A 0.000,B 0.000,C 90.000,E1 288.852} C_DIS
LIN {X -0.245,Y -637.585,Z 1000.404,A 0.000,B 0.000,C 90.000,E1 288.779} C_DIS
LIN {X 0.316,Y -637.576,Z 1000.404,A 0.000,B 0.000,C 90.000,E1 288.725} C_DIS
LIN {X -0.027,Y -637.986,Z 1000.403,A 0.000,B 0.000,C 90.000,E1 288.544} C_DIS
LIN {X -0.189,Y -640.036,Z 1000.401,A 0.000,B 0.000,C 90.000,E1 288.181} C_DIS
LIN {X -0.007,Y -647.084,Z 1000.395,A 0.000,B 0.000,C 90.000,E1 287.040} C_DIS
LIN {X -0.267,Y -650.613,Z 1000.391,A 0.000,B 0.000,C 90.000,E1 286.441} C_DIS
LIN {X 0.125,Y -653.660,Z 1000.388,A 0.000,B 0.000,C 90.000,E1 285.788} C_DIS
LIN {X 0.057,Y -655.628,Z 1000.385,A 0.000,B 0.000,C 90.000,E1 285.300} C_DIS
LIN {X -0.176,Y -657.203,Z 1000.382,A 0.000,B 0.000,C 90.000,E1 284.828} C_DIS
LIN {X -0.288,Y -657.946,Z 1000.381,A 0.000,B 0.000,C 90.000,E1 284.592} C_DIS
LIN {X 0.030,Y -659.424,Z 1000.377,A 0.000,B 0.000,C 90.000,E1 283.828} C_DIS
LIN {X -0.174,Y -660.195,Z 1000.374,A 0.000,B 0.000,C 90.000,E1 283.355} C_DIS
LIN {X 0.269,Y -660.625,Z 1000.371,A 0.000,B 0.000,C 90.000,E1 282.827} C_DIS
LIN {X -0.027,Y -660.881,Z 1000.367,A 0.000,B 0.000,C 90.000,E1 282.119} C_DIS
LIN {X -0.361,Y -660.842,Z 1000.365,A 0.000,B 0.000,C 90.000,E1 281.658} C_DIS
LIN {X 0.090,Y -660.597,Z 1000.362,A 0.000,B 0.000,C 90.000,E1 281.130} C_DIS
LIN {X -0.218,Y -659.773,Z 1000.358,A 0.000,B 0.000,C 90.000,E1 280.423} C_DIS
LIN {X 0.102,Y -658.918,Z 1000.355,A 0.000,B 0.000,C 90.000,E1 279.905} C_DIS
LIN {X -0.119,Y -657.854,Z 1000.352,A 0.000,B 0.000,C 90.000,E1 279.434} C_DIS
LIN {X 0.193,Y -656.413,Z 1000.350,A 0.000,B 0.000,C 90.000,E1 278.916} C_DIS
LIN {X -0.148,Y -654.619,Z 1000.347,A 0.000,B 0.000,C 90.000,E1 278.454} C_DIS
LIN {X -0.274,Y -653.622,Z 1000.346,A 0.000,B 0.000,C 90.000,E1 278.219} C_DIS
LIN {X 0.016,Y -651.310,Z 1000.343,A 0.000,B 0.000,C 90.000,E1 277.701} C_DIS
LIN {X 0.174,Y -647.589,Z 1000.339,A 0.000,B 0.000,C 90.000,E1 277.068} C_DIS
LIN {X -0.219,Y -644.038,Z 1000.337,A 0.000,B 0.000,C 90.000,E1 276.606} C_DIS
LIN {X 0.006,Y -639.973,Z 1000.334,A 0.000,B 0.000,C 90.000,E1 276.087} C_DIS
LIN {X 0.072,Y -634.203,Z 1000.330,A 0.000,B 0.000,C 90.000,E1 275.454} C_DIS
LIN {X -0.256,Y -629.078,Z 1000.328,A 0.000,B 0.000,C 90.000,E1 274.992} C_DIS
LIN {X -0.217,Y -622.426,Z 1000.324,A 0.000,B 0.000,C 90.000,E1 274.416} C_DIS
LIN {X -0.152,Y -618.177,Z 1000.323,A 0.000,B 0.000,C 90.000,E1 274.073} C_DIS
LIN {X 0.230,Y -612.161,Z 1000.320,A 0.000,B 0.000,C 90.000,E1 273.612} C_DIS
LIN {X 0.258,Y -605.891,Z 1000.318,A 0.000,B 0.000,C 90.000,E1 273.212} C_DIS
LIN {X -0.009,Y -599.326,Z 1000.316,A 0.000,B 0.000,C 90.000,E1 272.865} C_DIS
LIN {X 0.122,Y -592.325,Z 1000.314,A 0.000,B 0.000,C 90.000,E1 272.522} C_DIS
LIN {X -0.282,Y -588.280,Z 1000.313,A 0.000,B 0.000,C 90.000,E1 272.407} C_DIS
LIN {X 0.211,Y -584.834,Z 1000.313,A 0.000,B 0.000,C 90.000,E1 272.236} C_DIS
LIN {X 0.197,Y -576.977,Z 1000.311,A 0.000,B 0.000,C 90.000,E1 272.007} C_DIS
LIN {X -0.046,Y -571.193,Z 1000.311,A 0.000,B 0.000,C 90.000,E1 271.892} C_DIS
LIN {X 0.030,Y -565.225,Z 1000.310,A 0.000,B 0.000,C 90.000,E1 271.776} C_DIS
LIN {X -0.004,Y -558.312,Z 1000.310,A 0.000,B 0.000,C 90.000,E1 271.718} C_DIS
LIN {X -0.051,Y -543.566,Z 1000.310,A 0.000,B 0.000,C 90.000,E1 271.718} C_DIS
LIN {X 0.142,Y -543.164,Z 1000.309,A 0.000,B 0.000,C 90.000,E1 271.604} C_DIS
LIN {X -0.163,Y -542.932,Z 1000.309,A 0.000,B 0.000,C 90.000,E1 271.547} C_DIS
LIN {X -0.173,Y -542.123,Z 1000.304,A 0.000,B 0.000,C 90.000,E1 270.802} C_DIS
LIN {X 0.005,Y -540.757,Z 1000.293,A 0.000,B 0.000,C 90.000,E1 268.797} C_DIS
LIN {X 0.105,Y -540.000,Z 1000.287,A 0.000,B 0.000,C 90.000,E1 267.650} C_DIS
LIN {X 0.217,Y -538.754,Z 1000.278,A 0.000,B 0.000,C 90.000,E1 265.931} C_DIS
LIN {X -0.161,Y -537.620,Z 1000.270,A 0.000,B 0.000,C 90.000,E1 264.546} C_DIS
LIN {X -0.071,Y -536.392,Z 1000.262,A 0.000,B 0.000,C 90.000,E1 263.109} C_DIS
LIN {X 0.124,Y -535.021,Z 1000.254,A 0.000,B 0.000,C 90.000,E1 261.659} C_DIS
LIN {X 0.209,Y -533.553,Z 1000.246,A 0.000,B 0.000,C 90.000,E1 260.218} C_DIS
LIN {X -0.035,Y -531.741,Z 1000.236,A 0.000,B 0.000,C 90.000,E1 258.522} C_DIS
LIN {X 0.166,Y -530.202,Z 1000.228,A 0.000,B 0.000,C 90.000,E1 257.061} C_DIS
LIN {X -0.063,Y -528.626,Z 1000.220,A 0.000,B 0.000,C 90.000,E1 255.644} C_DIS
LIN {X 0.174,Y -525.708,Z 1000.206,A 0.000,B 0.000,C 90.000,E1 253.015} C_DIS
LIN {X 0.008,Y -524.429,Z 1000.199,A 0.000,B 0.000,C 90.000,E1 251.873} C_DIS
LIN {X -0.181,Y -523.005,Z 1000.193,A 0.000,B 0.000,C 90.000,E1 250.732} C_DIS
LIN {X 0.089,Y -520.788,Z 1000.183,A 0.000,B 0.000,C 90.000,E1 248.954} C_DIS
LIN {X -0.176,Y -518.523,Z 1000.173,A 0.000,B 0.000,C 90.000,E1 247.230} C_DIS
LIN {X -0.227,Y -517.339,Z 1000.169,A 0.000,B 0.000,C 90.000,E1 246.357} C_DIS
LIN {X -0.038,Y -514.256,Z 1000.157,A 0.000,B 0.000,C 90.000,E1 244.280} C_DIS
LIN {X 0.178,Y -511.413,Z 1000.147,A 0.000,B 0.000,C 90.000,E1 242.487} C_DIS
LIN {X -0.215,Y -509.078,Z 1000.139,A 0.000,B 0.000,C 90.000,E1 241.051} C_DIS
LIN {X 0.042,Y -506.508,Z 1000.131,A 0.000,B 0.000,C 90.000,E1 239.537} C_DIS
LIN {X 0.190,Y -504.260,Z 1000.124,A 0.000,B 0.000,C 90.000,E1 238.329} C_DIS
LIN {X 0.059,Y -500.646,Z 1000.114,A 0.000,B 0.000,C 90.000,E1 236.548} C_DIS
LIN {X 0.108,Y -497.967,Z 1000.108,A 0.000,B 0.000,C 90.000,E1 235.341} C_DIS
LIN {X -0.287,Y -495.917,Z 1000.103,A 0.000,B 0.000,C 90.000,E1 234.482} C_DIS
LIN {X -0.006,Y -493.709,Z 1000.098,A 0.000,B 0.000,C 90.000,E1 233.543} C_DIS
LIN {X 0.165,Y -487.762,Z 1000.084,A 0.000,B 0.000,C 90.000,E1 231.090} C_DIS
LIN {X -0.027,Y -485.581,Z 1000.079,A 0.000,B 0.000,C 90.000,E1 230.194} C_DIS
LIN {X 0.069,Y -482.072,Z 1000.070,A 0.000,B 0.000,C 90.000,E1 228.647} C_DIS
LIN {X -0.062,Y -475.378,Z 1000.053,A 0.000,B 0.000,C 90.000,E1 225.567} C_DIS
LIN {X -0.221,Y -472.130,Z 1000.044,A 0.000,B 0.000,C 90.000,E1 224.028} C_DIS
LIN {X -0.186,Y -469.437,Z 1000.038,A 0.000,B 0.000,C 90.000,E1 222.771} C_DIS
LIN {X -0.021,Y -465.288,Z 1000.027,A 0.000,B 0.000,C 90.000,E1 220.862} C_DIS
LIN {X -0.154,Y -463.157,Z 1000.022,A 0.000,B 0.000,C 90.000,E1 219.930} C_DIS
LIN {X 0.142,Y -460.286,Z 1000.015,A 0.000,B 0.000,C 90.000,E1 218.624} C_DIS
LIN {X -0.130,Y -455.419,Z 1000.002,A 0.000,B 0.000,C 90.000,E1 216.423} C_DIS
LIN {X -0.053,Y -451.179,Z 999.992,A 0.000,B 0.000,C 90.000,E1 214.485} C_DIS
LIN {X -0.144,Y -447.708,Z 999.983,A 0.000,B 0.000,C 90.000,E1 212.880} C_DIS
LIN {X -0.114,Y -443.485,Z 999.972,A 0.000,B 0.000,C 90.000,E1 210.924} C_DIS
LIN {X -0.071,Y -439.859,Z 999.963,A 0.000,B 0.000,C 90.000,E1 209.283} C_DIS
LIN {X -0.075,Y -435.331,Z 999.952,A 0.000,B 0.000,C 90.000,E1 207.308} C_DIS
LIN {X -0.020,Y -432.414,Z 999.944,A 0.000,B 0.000,C 90.000,E1 205.976} C_DIS
LIN {X -0.008,Y -429.349,Z 999.937,A 0.000,B 0.000,C 90.000,E1 204.643} C_DIS
LIN {X 0.124,Y -424.129,Z 999.924,A 0.000,B 0.000,C 90.000,E1 202.280} C_DIS
LIN {X 0.125,Y -418.361,Z 999.909,A 0.000,B 0.000,C 90.000,E1 199.577} C_DIS
LIN {X -0.180,Y -411.902,Z 999.890,A 0.000,B 0.000,C 90.000,E1 196.205} C_DIS
LIN {X -0.148,Y -408.922,Z 999.880,A 0.000,B 0.000,C 90.000,E1 194.481} C_DIS
LIN {X 0.107,Y -406.684,Z 999.873,A 0.000,B 0.000,C 90.000,E1 193.063} C_DIS
LIN {X -0.157,Y -403.914,Z 999.863,A 0.000,B 0.000,C 90.000,E1 191.366} C_DIS
LIN {X -0.107,Y -399.702,Z 999.848,A 0.000,B 0.000,C 90.000,E1 188.568} C_DIS
LIN {X -0.207,Y -398.780,Z 999.842,A 0.000,B 0.000,C 90.000,E1 187.530} C_DIS
LIN {X 0.171,Y -398.661,Z 999.840,A 0.000,B 0.000,C 90.000,E1 187.125} C_DIS
LIN {X 0.150,Y -398.730,Z 999.838,A 0.000,B 0.000,C 90.000,E1 186.777} C_DIS
LIN {X 0.072,Y -399.389,Z 999.833,A 0.000,B 0.000,C 90.000,E1 185.910} C_DIS
LIN {X 0.042,Y -399.640,Z 999.832,A 0.000,B 0.000,C 90.000,E1 185.739} C_DIS
LIN {X -0.195,Y -401.129,Z 999.829,A 0.000,B 0.000,C 90.000,E1 185.163} C_DIS
LIN {X 0.185,Y -402.272,Z 999.827,A 0.000,B 0.000,C 90.000,E1 184.759} C_DIS
LIN {X 0.135,Y -403.763,Z 999.825,A 0.000,B 0.000,C 90.000,E1 184.416} C_DIS
LIN {X 0.107,Y -407.320,Z 999.821,A 0.000,B 0.000,C 90.000,E1 183.784} C_DIS
LIN {X -0.144,Y -411.812,Z 999.818,A 0.000,B 0.000,C 90.000,E1 183.212} C_DIS
LIN {X 0.032,Y -418.942,Z 999.813,A 0.000,B 0.000,C 90.000,E1 182.350} C_DIS
LIN {X -0.023,Y -428.962,Z 999.807,A 0.000,B 0.000,C 90.000,E1 181.260} C_DIS
LIN {X 0.092,Y -443.174,Z 999.799,A 0.000,B 0.000,C 90.000,E1 179.714} C_DIS
LIN {X 0.014,Y -454.345,Z 999.792,A 0.000,B 0.000,C 90.000,E1 178.511} C_DIS
LIN {X 0.089,Y -462.519,Z 999.787,A 0.000,B 0.000,C 90.000,E1 177.593} C_DIS
LIN {X 0.144,Y -470.304,Z 999.782,A 0.000,B 0.000,C 90.000,E1 176.674} C_DIS
LIN {X 0.158,Y -475.521,Z 999.778,A 0.000,B 0.000,C 90.000,E1 176.045} C_DIS
LIN {X -0.134,Y -482.163,Z 999.773,A 0.000,B 0.000,C 90.000,E1 175.241} C_DIS
LIN {X 0.010,Y -490.001,Z 999.768,A 0.000,B 0.000,C 90.000,E1 174.147} C_DIS
LIN {X 0.075,Y -497.235,Z 999.762,A 0.000,B 0.000,C 90.000,E1 173.109} C_DIS
LIN {X 0.177,Y -505.441,Z 999.755,A 0.000,B 0.000,C 90.000,E1 171.894} C_DIS
LIN {X 0.214,Y -512.478,Z 999.749,A 0.000,B 0.000,C 90.000,E1 170.849} C_DIS
LIN {X -0.164,Y -520.849,Z 999.742,A 0.000,B 0.000,C 90.000,E1 169.567} C_DIS
LIN {X 0.054,Y -525.178,Z 999.738,A 0.000,B 0.000,C 90.000,E1 168.814} C_DIS
LIN {X -0.070,Y -531.387,Z 999.732,A 0.000,B 0.000,C 90.000,E1 167.813} C_DIS
LIN {X 0.180,Y -539.983,Z 999.724,A 0.000,B 0.000,C 90.000,E1 166.353} C_DIS
LIN {X 0.129,Y -550.594,Z 999.714,A 0.000,B 0.000,C 90.000,E1 164.519} C_DIS
LIN {X 0.091,Y -553.001,Z 999.712,A 0.000,B 0.000,C 90.000,E1 164.102} C_DIS
LIN {X 0.055,Y -559.801,Z 999.705,A 0.000,B 0.000,C 90.000,E1 162.851} C_DIS
LIN {X 0.086,Y -567.924,Z 999.696,A 0.000,B 0.000,C 90.000,E1 161.329} C_DIS
LIN {X 0.014,Y -573.438,Z 999.690,A 0.000,B 0.000,C 90.000,E1 160.242} C_DIS
LIN {X 0.011,Y -578.745,Z 999.684,A 0.000,B 0.000,C 90.000,E1 159.156} C_DIS
LIN {X 0.097,Y -582.541,Z 999.680,A 0.000,B 0.000,C 90.000,E1 158.337} C_DIS
LIN {X 0.072,Y -588.455,Z 999.672,A 0.000,B 0.000,C 90.000,E1 156.997} C_DIS
LIN {X 0.266,Y -591.764,Z 999.668,A 0.000,B 0.000,C 90.000,E1 156.177} C_DIS
LIN {X -0.040,Y -594.881,Z 999.663,A 0.000,B 0.000,C 90.000,E1 155.409} C_DIS
LIN {X 0.148,Y -598.646,Z 999.658,A 0.000,B 0.000,C 90.000,E1 154.332} C_DIS
LIN {X -0.006,Y -600.379,Z 999.655,A 0.000,B 0.000,C 90.000,E1 153.819} C_DIS
LIN {X 0.320,Y -602.803,Z 999.650,A 0.000,B 0.000,C 90.000,E1 152.999} C_DIS
LIN {X 0.012,Y -606.749,Z 999.643,A 0.000,B 0.000,C 90.000,E1 151.719} C_DIS
LIN {X 0.097,Y -609.727,Z 999.637,A 0.000,B 0.000,C 90.000,E1 150.667} C_DIS
LIN {X -0.343,Y -613.471,Z 999.630,A 0.000,B 0.000,C 90.000,E1 149.410} C_DIS
LIN {X 0.118,Y -617.028,Z 999.623,A 0.000,B 0.000,C 90.000,E1 148.074} C_DIS
LIN {X -0.088,Y -621.160,Z 999.614,A 0.000,B 0.000,C 90.000,E1 146.548} C_DIS
LIN {X -0.220,Y -626.143,Z 999.604,A 0.000,B 0.000,C 90.000,E1 144.769} C_DIS
LIN {X 0.290,Y -628.941,Z 999.599,A 0.000,B 0.000,C 90.000,E1 143.703} C_DIS
LIN {X 0.187,Y -633.084,Z 999.590,A 0.000,B 0.000,C 90.000,E1 142.190} C_DIS
LIN {X -0.221,Y -636.526,Z 999.583,A 0.000,B 0.000,C 90.000,E1 140.964} C_DIS
LIN {X -0.277,Y -640.571,Z 999.575,A 0.000,B 0.000,C 90.000,E1 139.461} C_DIS
LIN {X 0.176,Y -644.464,Z 999.566,A 0.000,B 0.000,C 90.000,E1 137.919} C_DIS
LIN {X -0.324,Y -649.938,Z 999.555,A 0.000,B 0.000,C 90.000,E1 135.972} C_DIS
LIN {X 0.301,Y -654.297,Z 999.547,A 0.000,B 0.000,C 90.000,E1 134.433} C_DIS
LIN {X 0.083,Y -659.029,Z 999.539,A 0.000,B 0.000,C 90.000,E1 132.975} C_DIS
LIN {X -0.033,Y -664.836,Z 999.529,A 0.000,B 0.000,C 90.000,E1 131.272} C_DIS
LIN {X -0.014,Y -668.086,Z 999.524,A 0.000,B 0.000,C 90.000,E1 130.297} C_DIS
LIN {X 0.143,Y -672.049,Z 999.517,A 0.000,B 0.000,C 90.000,E1 129.072} C_DIS
LIN {X -0.151,Y -675.627,Z 999.510,A 0.000,B 0.000,C 90.000,E1 127.890} C_DIS
LIN {X 0.151,Y -679.821,Z 999.502,A 0.000,B 0.000,C 90.000,E1 126.423} C_DIS
LIN {X 0.103,Y -683.175,Z 999.496,A 0.000,B 0.000,C 90.000,E1 125.231} C_DIS
LIN {X 0.107,Y -686.467,Z 999.489,A 0.000,B 0.000,C 90.000,E1 124.040} C_DIS
LIN {X 0.146,Y -688.910,Z 999.484,A 0.000,B 0.000,C 90.000,E1 123.086} C_DIS
LIN {X 0.084,Y -692.540,Z 999.476,A 0.000,B 0.000,C 90.000,E1 121.671} C_DIS
LIN {X 0.201,Y -694.894,Z 999.471,A 0.000,B 0.000,C 90.000,E1 120.718} C_DIS
LIN {X 0.340,Y -696.493,Z 999.467,A 0.000,B 0.000,C 90.000,E1 120.001} C_DIS
LIN {X 0.242,Y -697.484,Z 999.464,A 0.000,B 0.000,C 90.000,E1 119.539} C_DIS
LIN {X 0.062,Y -699.030,Z 999.459,A 0.000,B 0.000,C 90.000,E1 118.615} C_DIS
LIN {X 0.245,Y -699.945,Z 999.455,A 0.000,B 0.000,C 90.000,E1 117.897} C_DIS
LIN {X -0.160,Y -700.373,Z 999.453,A 0.000,B 0.000,C 90.000,E1 117.462} C_DIS
LIN {X 0.200,Y -701.723,Z 999.443,A 0.000,B 0.000,C 90.000,E1 115.796} C_DIS
LIN {X 0.100,Y -702.205,Z 999.440,A 0.000,B 0.000,C 90.000,E1 115.103} C_DIS
LIN {X 0.019,Y -702.452,Z 999.437,A 0.000,B 0.000,C 90.000,E1 114.643} C_DIS
LIN {X -0.355,Y -702.510,Z 999.434,A 0.000,B 0.000,C 90.000,E1 114.207} C_DIS
LIN {X 0.198,Y -701.966,Z 999.432,A 0.000,B 0.000,C 90.000,E1 113.695} C_DIS
LIN {X 0.192,Y -701.546,Z 999.430,A 0.000,B 0.000,C 90.000,E1 113.462} C_DIS
LIN {X -0.049,Y -698.860,Z 999.427,A 0.000,B 0.000,C 90.000,E1 112.898} C_DIS
LIN {X 0.083,Y -698.050,Z 999.427,A 0.000,B 0.000,C 90.000,E1 112.770} C_DIS
LIN {X 0.214,Y -696.848,Z 999.426,A 0.000,B 0.000,C 90.000,E1 112.642} C_DIS
LIN {X -0.081,Y -692.585,Z 999.424,A 0.000,B 0.000,C 90.000,E1 112.333} C_DIS
LIN {X 0.226,Y -691.195,Z 999.424,A 0.000,B 0.000,C 90.000,E1 112.206} C_DIS
LIN {X -0.367,Y -689.134,Z 999.423,A 0.000,B 0.000,C 90.000,E1 112.153} C_DIS
LIN {X -0.079,Y -684.542,Z 999.422,A 0.000,B 0.000,C 90.000,E1 111.972} C_DIS
LIN {X -0.236,Y -679.444,Z 999.422,A 0.000,B 0.000,C 90.000,E1 111.897} C_DIS
LIN {X -0.347,Y -674.963,Z 999.421,A 0.000,B 0.000,C 90.000,E1 111.844} C_DIS
LIN {X -0.367,Y -619.272,Z 999.421,A 0.000,B 0.000,C 90.000,E1 111.844} C_DIS
LIN {X 0.186,Y -615.528,Z 999.421,A 0.000,B 0.000,C 90.000,E1 111.716} C_DIS
LIN {X -0.087,Y -610.080,Z 999.420,A 0.000,B 0.000,C 90.000,E1 111.589} C_DIS
LIN {X -0.272,Y -602.122,Z 999.418,A 0.000,B 0.000,C 90.000,E1 111.280} C_DIS
LIN {X 0.199,Y -597.201,Z 999.417,A 0.000,B 0.000,C 90.000,E1 110.972} C_DIS
LIN {X 0.220,Y -594.218,Z 999.416,A 0.000,B 0.000,C 90.000,E1 110.791} C_DIS
LIN {X -0.013,Y -589.545,Z 999.414,A 0.000,B 0.000,C 90.000,E1 110.482} C_DIS
LIN {X 0.140,Y -577.569,Z 999.409,A 0.000,B 0.000,C 90.000,E1 109.504} C_DIS
LIN {X 0.356,Y -573.221,Z 999.407,A 0.000,B 0.000,C 90.000,E1 109.141} C_DIS
LIN {X -0.101,Y -569.582,Z 999.405,A 0.000,B 0.000,C 90.000,E1 108.960} C_DIS
LIN {X -0.014,Y -564.829,Z 999.404,A 0.000,B 0.000,C 90.000,E1 108.671} C_DIS
LIN {X 0.162,Y -550.750,Z 999.400,A 0.000,B 0.000,C 90.000,E1 107.946} C_DIS
LIN {X 0.066,Y -549.858,Z 999.399,A 0.000,B 0.000,C 90.000,E1 107.873} C_DIS
LIN {X 0.146,Y -548.990,Z 999.399,A 0.000,B 0.000,C 90.000,E1 107.764} C_DIS
LIN {X 0.118,Y -548.975,Z 999.399,A 0.000,B 0.000,C 90.000,E1 107.764} C_DIS
LIN {X -0.316,Y -548.634,Z 999.398,A 0.000,B 0.000,C 90.000,E1 107.583} C_DIS
LIN {X 0.274,Y -548.538,Z 999.394,A 0.000,B 0.000,C 90.000,E1 106.913} C_DIS
LIN {X -0.248,Y -549.057,Z 999.388,A 0.000,B 0.000,C 90.000,E1 105.843} C_DIS
LIN {X 0.223,Y -550.021,Z 999.377,A 0.000,B 0.000,C 90.000,E1 103.828} C_DIS
LIN {X 0.101,Y -552.995,Z 999.357,A 0.000,B 0.000,C 90.000,E1 100.197} C_DIS
LIN {X -0.227,Y -555.129,Z 999.346,A 0.000,B 0.000,C 90.000,E1 98.276} C_DIS
LIN {X 0.250,Y -556.613,Z 999.338,A 0.000,B 0.000,C 90.000,E1 96.834} C_DIS
LIN {X 0.076,Y -557.645,Z 999.332,A 0.000,B 0.000,C 90.000,E1 95.739} C_DIS
LIN {X -0.210,Y -558.308,Z 999.327,A 0.000,B 0.000,C 90.000,E1 94.935} C_DIS
LIN {X 0.276,Y -559.217,Z 999.320,A 0.000,B 0.000,C 90.000,E1 93.498} C_DIS
LIN {X 0.095,Y -559.851,Z 999.313,A 0.000,B 0.000,C 90.000,E1 92.407} C_DIS
LIN {X -0.268,Y -560.950,Z 999.301,A 0.000,B 0.000,C 90.000,E1 90.229} C_DIS
LIN {X 0.216,Y -561.540,Z 999.294,A 0.000,B 0.000,C 90.000,E1 88.797} C_DIS
LIN {X 0.063,Y -561.857,Z 999.287,A 0.000,B 0.000,C 90.000,E1 87.707} C_DIS
LIN {X 0.107,Y -562.114,Z 999.278,A 0.000,B 0.000,C 90.000,E1 86.045} C_DIS
LIN {X -0.237,Y -562.406,Z 999.267,A 0.000,B 0.000,C 90.000,E1 84.147} C_DIS
LIN {X 0.045,Y -562.746,Z 999.257,A 0.000,B 0.000,C 90.000,E1 82.186} C_DIS
LIN {X -0.148,Y -563.260,Z 999.246,A 0.000,B 0.000,C 90.000,E1 80.274} C_DIS
LIN {X -0.123,Y -564.087,Z 999.235,A 0.000,B 0.000,C 90.000,E1 78.342} C_DIS
LIN {X -0.234,Y -564.940,Z 999.226,A 0.000,B 0.000,C 90.000,E1 76.700} C_DIS
LIN {X -0.036,Y -566.184,Z 999.215,A 0.000,B 0.000,C 90.000,E1 74.755} C_DIS
LIN {X 0.166,Y -567.379,Z 999.206,A 0.000,B 0.000,C 90.000,E1 73.087} C_DIS
LIN {X -0.317,Y -568.437,Z 999.199,A 0.000,B 0.000,C 90.000,E1 71.764} C_DIS
LIN {X 0.283,Y -569.564,Z 999.189,A 0.000,B 0.000,C 90.000,E1 70.061} C_DIS
LIN {X -0.158,Y -570.512,Z 999.180,A 0.000,B 0.000,C 90.000,E1 68.465} C_DIS
LIN {X 0.161,Y -571.338,Z 999.171,A 0.000,B 0.000,C 90.000,E1 66.794} C_DIS
LIN {X -0.224,Y -571.823,Z 999.165,A 0.000,B 0.000,C 90.000,E1 65.741} C_DIS
LIN {X 0.228,Y -572.390,Z 999.158,A 0.000,B 0.000,C 90.000,E1 64.332} C_DIS
LIN {X -0.068,Y -572.802,Z 999.150,A 0.000,B 0.000,C 90.000,E1 62.999} C_DIS
LIN {X -0.266,Y -573.266,Z 999.141,A 0.000,B 0.000,C 90.000,E1 61.385} C_DIS
LIN {X -0.182,Y -573.673,Z 999.132,A 0.000,B 0.000,C 90.000,E1 59.744} C_DIS
LIN {X 0.364,Y -573.915,Z 999.124,A 0.000,B 0.000,C 90.000,E1 58.329} C_DIS
LIN {X 0.261,Y -574.131,Z 999.115,A 0.000,B 0.000,C 90.000,E1 56.707} C_DIS
LIN {X -0.146,Y -574.305,Z 999.108,A 0.000,B 0.000,C 90.000,E1 55.388} C_DIS
LIN {X 0.103,Y -574.233,Z 999.102,A 0.000,B 0.000,C 90.000,E1 54.276} C_DIS
LIN {X -0.262,Y -574.169,Z 999.097,A 0.000,B 0.000,C 90.000,E1 53.497} C_DIS
LIN {X 0.174,Y -573.952,Z 999.093,A 0.000,B 0.000,C 90.000,E1 52.637} C_DIS
LIN {X 0.296,Y -573.396,Z 999.087,A 0.000,B 0.000,C 90.000,E1 51.537} C_DIS
LIN {X 0.111,Y -572.604,Z 999.079,A 0.000,B 0.000,C 90.000,E1 50.194} C_DIS
LIN {X -0.089,Y -571.455,Z 999.071,A 0.000,B 0.000,C 90.000,E1 48.852} C_DIS
LIN {X -0.059,Y -570.367,Z 999.065,A 0.000,B 0.000,C 90.000,E1 47.757} C_DIS
LIN {X -0.127,Y -569.363,Z 999.061,A 0.000,B 0.000,C 90.000,E1 46.944} C_DIS
LIN {X 0.261,Y -567.623,Z 999.055,A 0.000,B 0.000,C 90.000,E1 45.810} C_DIS
LIN {X 0.139,Y -566.115,Z 999.050,A 0.000,B 0.000,C 90.000,E1 45.000} C_DIS
LIN {X -0.314,Y -563.867,Z 999.044,A 0.000,B 0.000,C 90.000,E1 43.947} C_DIS
LIN {X -0.068,Y -561.923,Z 999.039,A 0.000,B 0.000,C 90.000,E1 43.095} C_DIS
LIN {X 0.075,Y -560.465,Z 999.036,A 0.000,B 0.000,C 90.000,E1 42.528} C_DIS
LIN {X 0.019,Y -556.265,Z 999.029,A 0.000,B 0.000,C 90.000,E1 41.148} C_DIS
LIN {X -0.181,Y -553.313,Z 999.024,A 0.000,B 0.000,C 90.000,E1 40.334} C_DIS
LIN {X -0.117,Y -551.182,Z 999.021,A 0.000,B 0.000,C 90.000,E1 39.769} C_DIS
LIN {X 0.055,Y -547.640,Z 999.016,A 0.000,B 0.000,C 90.000,E1 38.910} C_DIS
LIN {X -0.086,Y -544.470,Z 999.012,A 0.000,B 0.000,C 90.000,E1 38.222} C_DIS
LIN {X -0.141,Y -539.722,Z 999.007,A 0.000,B 0.000,C 90.000,E1 37.237} C_DIS
LIN {X -0.085,Y -533.840,Z 999.000,A 0.000,B 0.000,C 90.000,E1 36.091} C_DIS
LIN {X -0.103,Y -529.110,Z 998.996,A 0.000,B 0.000,C 90.000,E1 35.231} C_DIS
LIN {X 0.285,Y -525.744,Z 998.992,A 0.000,B 0.000,C 90.000,E1 34.612} C_DIS
LIN {X -0.122,Y -520.457,Z 998.988,A 0.000,B 0.000,C 90.000,E1 33.785} C_DIS
LIN {X 0.025,Y -515.734,Z 998.984,A 0.000,B 0.000,C 90.000,E1 33.038} C_DIS
LIN {X 0.223,Y -509.628,Z 998.979,A 0.000,B 0.000,C 90.000,E1 32.133} C_DIS
LIN {X 0.186,Y -505.235,Z 998.975,A 0.000,B 0.000,C 90.000,E1 31.544} C_DIS
LIN {X -0.103,Y -499.341,Z 998.971,A 0.000,B 0.000,C 90.000,E1 30.846} C_DIS
LIN {X -0.011,Y -495.500,Z 998.969,A 0.000,B 0.000,C 90.000,E1 30.384} C_DIS
LIN {X 0.234,Y -486.011,Z 998.963,A 0.000,B 0.000,C 90.000,E1 29.333} C_DIS
LIN {X 0.143,Y -475.992,Z 998.958,A 0.000,B 0.000,C 90.000,E1 28.359} C_DIS
LIN {X 0.252,Y -465.831,Z 998.952,A 0.000,B 0.000,C 90.000,E1 27.385} C_DIS
LIN {X -0.045,Y -458.314,Z 998.949,A 0.000,B 0.000,C 90.000,E1 26.744} C_DIS
LIN {X 0.164,Y -446.034,Z 998.943,A 0.000,B 0.000,C 90.000,E1 25.668} C_DIS
LIN {X 0.160,Y -434.154,Z 998.937,A 0.000,B 0.000,C 90.000,E1 24.643} C_DIS
LIN {X -0.242,Y -419.362,Z 998.930,A 0.000,B 0.000,C 90.000,E1 23.334} C_DIS
LIN {X 0.065,Y -406.419,Z 998.922,A 0.000,B 0.000,C 90.000,E1 21.972} C_DIS
LIN {X -0.189,Y -399.414,Z 998.918,A 0.000,B 0.000,C 90.000,E1 21.227} C_DIS
LIN {X 0.091,Y -396.777,Z 998.916,A 0.000,B 0.000,C 90.000,E1 20.865} C_DIS
LIN {X 0.002,Y -393.114,Z 998.913,A 0.000,B 0.000,C 90.000,E1 20.301} C_DIS
LIN {X 0.060,Y -391.688,Z 998.911,A 0.000,B 0.000,C 90.000,E1 19.939} C_DIS
LIN {X 0.141,Y -390.873,Z 998.909,A 0.000,B 0.000,C 90.000,E1 19.577} C_DIS
LIN {X 0.056,Y -390.374,Z 998.907,A 0.000,B 0.000,C 90.000,E1 19.322} C_DIS
LIN {X 0.064,Y -390.353,Z 998.904,A 0.000,B 0.000,C 90.000,E1 18.779} C_DIS
LIN {X 0.147,Y -390.717,Z 998.900,A 0.000,B 0.000,C 90.000,E1 18.055} C_DIS
LIN {X -0.135,Y -393.858,Z 998.883,A 0.000,B 0.000,C 90.000,E1 14.898} C_DIS
LIN {X -0.100,Y -399.482,Z 998.859,A 0.000,B 0.000,C 90.000,E1 10.658} C_DIS
LIN {X 0.170,Y -406.134,Z 998.838,A 0.000,B 0.000,C 90.000,E1 6.777} C_DIS
LIN {X 0.145,Y -412.619,Z 998.821,A 0.000,B 0.000,C 90.000,E1 3.669} C_DIS
LIN {X -0.200,Y -417.192,Z 998.809,A 0.000,B 0.000,C 90.000,E1 1.661} C_DIS
LIN {X -0.160,Y -419.533,Z 998.805,A 0.000,B 0.000,C 90.000,E1 0.974} C_DIS
LIN {X -0.146,Y -420.300,Z 998.804,A 0.000,B 0.000,C 90.000,E1 0.802} C_DIS
LIN {X -0.149,Y -423.377,Z 998.802,A 0.000,B 0.000,C 90.000,E1 0.286} C_DIS
LIN {X 0.162,Y -428.263,Z 998.799,A 0.000,B 0.000,C 90.000,E1 359.771} C_DIS
LIN {X 0.186,Y -432.571,Z 998.797,A 0.000,B 0.000,C 90.000,E1 359.484} C_DIS
LIN {X 0.133,Y -442.756,Z 998.794,A 0.000,B 0.000,C 90.000,E1 358.912} C_DIS
LIN {X 0.209,Y -452.826,Z 998.791,A 0.000,B 0.000,C 90.000,E1 358.339} C_DIS
LIN {X 0.216,Y -467.709,Z 998.786,A 0.000,B 0.000,C 90.000,E1 357.478} C_DIS
LIN {X -0.199,Y -482.667,Z 998.781,A 0.000,B 0.000,C 90.000,E1 356.674} C_DIS
LIN {X -0.144,Y -492.537,Z 998.778,A 0.000,B 0.000,C 90.000,E1 356.102} C_DIS
LIN {X -0.174,Y -502.295,Z 998.775,A 0.000,B 0.000,C 90.000,E1 355.527} C_DIS
LIN {X 0.059,Y -511.823,Z 998.772,A 0.000,B 0.000,C 90.000,E1 354.894} C_DIS
LIN {X -0.106,Y -519.530,Z 998.769,A 0.000,B 0.000,C 90.000,E1 354.375} C_DIS
LIN {X 0.094,Y -527.040,Z 998.766,A 0.000,B 0.000,C 90.000,E1 353.799} C_DIS
LIN {X 0.015,Y -534.349,Z 998.762,A 0.000,B 0.000,C 90.000,E1 353.223} C_DIS
LIN {X -0.109,Y -538.451,Z 998.760,A 0.000,B 0.000,C 90.000,E1 352.875} C_DIS
LIN {X 0.133,Y -542.606,Z 998.758,A 0.000,B 0.000,C 90.000,E1 352.470} C_DIS
LIN {X -0.127,Y -549.149,Z 998.755,A 0.000,B 0.000,C 90.000,E1 351.837} C_DIS
LIN {X 0.266,Y -554.247,Z 998.752,A 0.000,B 0.000,C 90.000,E1 351.254} C_DIS
LIN {X 0.201,Y -559.997,Z 998.748,A 0.000,B 0.000,C 90.000,E1 350.566} C_DIS
LIN {X -0.059,Y -564.293,Z 998.745,A 0.000,B 0.000,C 90.000,E1 350.038} C_DIS
LIN {X 0.027,Y -568.980,Z 998.741,A 0.000,B 0.000,C 90.000,E1 349.342} C_DIS
LIN {X -0.168,Y -572.373,Z 998.738,A 0.000,B 0.000,C 90.000,E1 348.814} C_DIS
LIN {X -0.013,Y -576.362,Z 998.734,A 0.000,B 0.000,C 90.000,E1 348.117} C_DIS
LIN {X -0.046,Y -581.482,Z 998.729,A 0.000,B 0.000,C 90.000,E1 347.173} C_DIS
LIN {X -0.245,Y -586.947,Z 998.723,A 0.000,B 0.000,C 90.000,E1 346.117} C_DIS
LIN {X 0.035,Y -593.331,Z 998.715,A 0.000,B 0.000,C 90.000,E1 344.755} C_DIS
LIN {X 0.140,Y -598.072,Z 998.709,A 0.000,B 0.000,C 90.000,E1 343.685} C_DIS
LIN {X -0.095,Y -602.545,Z 998.704,A 0.000,B 0.000,C 90.000,E1 342.653} C_DIS
LIN {X 0.046,Y -607.837,Z 998.696,A 0.000,B 0.000,C 90.000,E1 341.329} C_DIS
LIN {X -0.307,Y -612.778,Z 998.689,A 0.000,B 0.000,C 90.000,E1 340.061} C_DIS
LIN {X -0.083,Y -615.350,Z 998.685,A 0.000,B 0.000,C 90.000,E1 339.263} C_DIS
LIN {X -0.084,Y -618.597,Z 998.679,A 0.000,B 0.000,C 90.000,E1 338.230} C_DIS
LIN {X 0.176,Y -622.502,Z 998.672,A 0.000,B 0.000,C 90.000,E1 336.922} C_DIS
LIN {X -0.074,Y -625.376,Z 998.666,A 0.000,B 0.000,C 90.000,E1 335.921} C_DIS
LIN {X -0.290,Y -628.009,Z 998.661,A 0.000,B 0.000,C 90.000,E1 334.921} C_DIS
LIN {X -0.204,Y -630.493,Z 998.655,A 0.000,B 0.000,C 90.000,E1 333.896} C_DIS
LIN {X -0.116,Y -632.147,Z 998.651,A 0.000,B 0.000,C 90.000,E1 333.127} C_DIS
LIN {X 0.105,Y -635.168,Z 998.642,A 0.000,B 0.000,C 90.000,E1 331.591} C_DIS
LIN {X 0.030,Y -637.013,Z 998.637,A 0.000,B 0.000,C 90.000,E1 330.589} C_DIS
LIN {X -0.381,Y -638.366,Z 998.633,A 0.000,B 0.000,C 90.000,E1 329.871} C_DIS
LIN {X 0.028,Y -640.687,Z 998.624,A 0.000,B 0.000,C 90.000,E1 328.329} C_DIS
LIN {X -0.020,Y -641.625,Z 998.620,A 0.000,B 0.000,C 90.000,E1 327.582} C_DIS
LIN {X -0.009,Y -642.857,Z 998.614,A 0.000,B 0.000,C 90.000,E1 326.580} C_DIS
LIN {X -0.165,Y -643.894,Z 998.609,A 0.000,B 0.000,C 90.000,E1 325.595} C_DIS
LIN {X 0.223,Y -644.734,Z 998.603,A 0.000,B 0.000,C 90.000,E1 324.562} C_DIS
LIN {X -0.007,Y -645.437,Z 998.596,A 0.000,B 0.000,C 90.000,E1 323.336} C_DIS
LIN {X -0.129,Y -645.968,Z 998.591,A 0.000,B 0.000,C 90.000,E1 322.351} C_DIS
LIN {X -0.002,Y -646.609,Z 998.581,A 0.000,B 0.000,C 90.000,E1 320.598} C_DIS
LIN {X -0.077,Y -647.534,Z 998.569,A 0.000,B 0.000,C 90.000,E1 318.366} C_DIS
LIN {X 0.068,Y -648.524,Z 998.560,A 0.000,B 0.000,C 90.000,E1 316.863} C_DIS
LIN {X -0.334,Y -649.512,Z 998.551,A 0.000,B 0.000,C 90.000,E1 315.162} C_DIS
LIN {X 0.157,Y -650.964,Z 998.540,A 0.000,B 0.000,C 90.000,E1 313.137} C_DIS
LIN {X -0.116,Y -651.982,Z 998.532,A 0.000,B 0.000,C 90.000,E1 311.676} C_DIS
LIN {X -0.317,Y -652.671,Z 998.525,A 0.000,B 0.000,C 90.000,E1 310.458} C_DIS
LIN {X -0.067,Y -653.361,Z 998.516,A 0.000,B 0.000,C 90.000,E1 308.955} C_DIS
LIN {X 0.296,Y -653.991,Z 998.508,A 0.000,B 0.000,C 90.000,E1 307.443} C_DIS
LIN {X -0.238,Y -654.289,Z 998.503,A 0.000,B 0.000,C 90.000,E1 306.503} C_DIS
LIN {X -0.243,Y -654.512,Z 998.495,A 0.000,B 0.000,C 90.000,E1 305.025} C_DIS
LIN {X -0.163,Y -654.857,Z 998.485,A 0.000,B 0.000,C 90.000,E1 303.293} C_DIS
LIN {X -0.201,Y -659.771,Z 998.453,A 0.000,B 0.000,C 90.000,E1 297.641} C_DIS
LIN {X -0.137,Y -661.517,Z 998.447,A 0.000,B 0.000,C 90.000,E1 296.411} C_DIS
LIN {X -0.201,Y -663.683,Z 998.439,A 0.000,B 0.000,C 90.000,E1 294.951} C_DIS
LIN {X 0.091,Y -664.942,Z 998.433,A 0.000,B 0.000,C 90.000,E1 293.951} C_DIS
LIN {X 0.257,Y -665.751,Z 998.429,A 0.000,B 0.000,C 90.000,E1 293.206} C_DIS
LIN {X -0.181,Y -666.266,Z 998.425,A 0.000,B 0.000,C 90.000,E1 292.514} C_DIS
LIN {X -0.147,Y -666.399,Z 998.422,A 0.000,B 0.000,C 90.000,E1 292.025} C_DIS
LIN {X -0.108,Y -666.080,Z 998.420,A 0.000,B 0.000,C 90.000,E1 291.535} C_DIS
LIN {X 0.033,Y -665.794,Z 998.418,A 0.000,B 0.000,C 90.000,E1 291.280} C_DIS
LIN {X 0.068,Y -664.039,Z 998.416,A 0.000,B 0.000,C 90.000,E1 290.791} C_DIS
LIN {X -0.034,Y -662.895,Z 998.414,A 0.000,B 0.000,C 90.000,E1 290.556} C_DIS
LIN {X 0.030,Y -661.908,Z 998.414,A 0.000,B 0.000,C 90.000,E1 290.429} C_DIS
LIN {X 0.113,Y -656.861,Z 998.411,A 0.000,B 0.000,C 90.000,E1 289.939} C_DIS
LIN {X 0.229,Y -655.145,Z 998.410,A 0.000,B 0.000,C 90.000,E1 289.812} C_DIS
LIN {X 0.029,Y -648.833,Z 998.408,A 0.000,B 0.000,C 90.000,E1 289.450} C_DIS
LIN {X 0.050,Y -642.506,Z 998.406,A 0.000,B 0.000,C 90.000,E1 289.087} C_DIS
LIN {X 0.080,Y -638.939,Z 998.405,A 0.000,B 0.000,C 90.000,E1 288.852} C_DIS
LIN {X 0.046,Y -638.908,Z 998.405,A 0.000,B 0.000,C 90.000,E1 288.852} C_DIS
LIN {X -0.223,Y -638.775,Z 998.405,A 0.000,B 0.000,C 90.000,E1 288.852} C_DIS
LIN {X -0.256,Y -638.770,Z 998.405,A 0.000,B 0.000,C 90.000,E1 288.852} C_DIS
LIN {X 0.368,Y -639.213,Z 998.404,A 0.000,B 0.000,C 90.000,E1 288.598} C_DIS
LIN {X 0.196,Y -640.358,Z 998.402,A 0.000,B 0.000,C 90.000,E1 288.362} C_DIS
LIN {X -0.091,Y -647.960,Z 998.395,A 0.000,B 0.000,C 90.000,E1 287.166} C_DIS
LIN {X -0.316,Y -652.170,Z 998.391,A 0.000,B 0.000,C 90.000,E1 286.441} C_DIS
LIN {X 0.211,Y -654.023,Z 998.389,A 0.000,B 0.000,C 90.000,E1 286.024} C_DIS
LIN {X 0.090,Y -655.141,Z 998.388,A 0.000,B 0.000,C 90.000,E1 285.788} C_DIS
LIN {X 0.030,Y -657.074,Z 998.385,A 0.000,B 0.000,C 90.000,E1 285.300} C_DIS
LIN {X -0.193,Y -658.643,Z 998.382,A 0.000,B 0.000,C 90.000,E1 284.828} C_DIS
LIN {X 0.337,Y -659.314,Z 998.381,A 0.000,B 0.000,C 90.000,E1 284.537} C_DIS
LIN {X 0.133,Y -660.350,Z 998.378,A 0.000,B 0.000,C 90.000,E1 284.064} C_DIS
LIN {X -0.164,Y -661.500,Z 998.374,A 0.000,B 0.000,C 90.000,E1 283.355} C_DIS
LIN {X 0.195,Y -662.054,Z 998.370,A 0.000,B 0.000,C 90.000,E1 282.591} C_DIS
LIN {X 0.005,Y -662.199,Z 998.367,A 0.000,B 0.000,C 90.000,E1 282.119} C_DIS
LIN {X -0.321,Y -662.162,Z 998.365,A 0.000,B 0.000,C 90.000,E1 281.658} C_DIS
LIN {X 0.139,Y -661.909,Z 998.362,A 0.000,B 0.000,C 90.000,E1 281.130} C_DIS
LIN {X -0.156,Y -661.141,Z 998.358,A 0.000,B 0.000,C 90.000,E1 280.423} C_DIS
LIN {X 0.173,Y -660.298,Z 998.355,A 0.000,B 0.000,C 90.000,E1 279.905} C_DIS
LIN {X -0.148,Y -659.235,Z 998.352,A 0.000,B 0.000,C 90.000,E1 279.443} C_DIS
LIN {X 0.283,Y -657.816,Z 998.350,A 0.000,B 0.000,C 90.000,E1 278.916} C_DIS
LIN {X -0.050,Y -656.060,Z 998.347,A 0.000,B 0.000,C 90.000,E1 278.454} C_DIS
LIN {X -0.172,Y -655.110,Z 998.346,A 0.000,B 0.000,C 90.000,E1 278.219} C_DIS
LIN {X 0.128,Y -652.837,Z 998.343,A 0.000,B 0.000,C 90.000,E1 277.701} C_DIS
LIN {X -0.346,Y -649.250,Z 998.339,A 0.000,B 0.000,C 90.000,E1 277.125} C_DIS
LIN {X -0.086,Y -645.800,Z 998.337,A 0.000,B 0.000,C 90.000,E1 276.606} C_DIS
LIN {X 0.097,Y -640.763,Z 998.333,A 0.000,B 0.000,C 90.000,E1 275.967} C_DIS
LIN {X 0.232,Y -636.216,Z 998.330,A 0.000,B 0.000,C 90.000,E1 275.454} C_DIS
LIN {X -0.179,Y -631.181,Z 998.328,A 0.000,B 0.000,C 90.000,E1 274.992} C_DIS
LIN {X 0.261,Y -625.872,Z 998.325,A 0.000,B 0.000,C 90.000,E1 274.473} C_DIS
LIN {X 0.295,Y -618.853,Z 998.322,A 0.000,B 0.000,C 90.000,E1 273.898} C_DIS
LIN {X 0.209,Y -611.267,Z 998.319,A 0.000,B 0.000,C 90.000,E1 273.383} C_DIS
LIN {X -0.259,Y -604.972,Z 998.317,A 0.000,B 0.000,C 90.000,E1 273.037} C_DIS
LIN {X 0.073,Y -598.288,Z 998.315,A 0.000,B 0.000,C 90.000,E1 272.636} C_DIS
LIN {X -0.293,Y -591.279,Z 998.313,A 0.000,B 0.000,C 90.000,E1 272.350} C_DIS
LIN {X -0.154,Y -585.306,Z 998.312,A 0.000,B 0.000,C 90.000,E1 272.121} C_DIS
LIN {X -0.120,Y -577.822,Z 998.310,A 0.000,B 0.000,C 90.000,E1 271.892} C_DIS
LIN {X 0.214,Y -572.118,Z 998.310,A 0.000,B 0.000,C 90.000,E1 271.718} C_DIS
LIN {X 0.142,Y -565.886,Z 998.309,A 0.000,B 0.000,C 90.000,E1 271.604} C_DIS
LIN {X -0.188,Y -563.270,Z 998.309,A 0.000,B 0.000,C 90.000,E1 271.604} C_DIS
LIN {X -0.024,Y -557.903,Z 998.309,A 0.000,B 0.000,C 90.000,E1 271.547} C_DIS
LIN {X -0.053,Y -543.183,Z 998.309,A 0.000,B 0.000,C 90.000,E1 271.547} C_DIS
LIN {X 0.025,Y -542.601,Z 998.306,A 0.000,B 0.000,C 90.000,E1 271.146} C_DIS
LIN {X 0.259,Y -540.739,Z 998.292,A 0.000,B 0.000,C 90.000,E1 268.568} C_DIS
LIN {X -0.165,Y -539.763,Z 998.284,A 0.000,B 0.000,C 90.000,E1 267.192} C_DIS
LIN {X -0.034,Y -538.700,Z 998.276,A 0.000,B 0.000,C 90.000,E1 265.755} C_DIS
LIN {X 0.031,Y -537.841,Z 998.270,A 0.000,B 0.000,C 90.000,E1 264.609} C_DIS
LIN {X 0.176,Y -536.599,Z 998.262,A 0.000,B 0.000,C 90.000,E1 263.166} C_DIS
LIN {X -0.180,Y -534.930,Z 998.253,A 0.000,B 0.000,C 90.000,E1 261.489} C_DIS
LIN {X -0.010,Y -533.475,Z 998.245,A 0.000,B 0.000,C 90.000,E1 260.038} C_DIS
LIN {X 0.272,Y -531.638,Z 998.235,A 0.000,B 0.000,C 90.000,E1 258.285} C_DIS
LIN {X -0.082,Y -530.403,Z 998.229,A 0.000,B 0.000,C 90.000,E1 257.173} C_DIS
LIN {X 0.212,Y -528.839,Z 998.221,A 0.000,B 0.000,C 90.000,E1 255.700} C_DIS
LIN {X -0.033,Y -525.616,Z 998.205,A 0.000,B 0.000,C 90.000,E1 252.834} C_DIS
LIN {X -0.200,Y -524.293,Z 998.198,A 0.000,B 0.000,C 90.000,E1 251.692} C_DIS
LIN {X -0.232,Y -522.454,Z 998.190,A 0.000,B 0.000,C 90.000,E1 250.242} C_DIS
LIN {X -0.125,Y -520.624,Z 998.182,A 0.000,B 0.000,C 90.000,E1 248.773} C_DIS
LIN {X 0.082,Y -518.369,Z 998.172,A 0.000,B 0.000,C 90.000,E1 246.997} C_DIS
LIN {X 0.232,Y -517.112,Z 998.167,A 0.000,B 0.000,C 90.000,E1 246.102} C_DIS
LIN {X -0.051,Y -514.897,Z 998.159,A 0.000,B 0.000,C 90.000,E1 244.665} C_DIS
LIN {X 0.071,Y -513.565,Z 998.154,A 0.000,B 0.000,C 90.000,E1 243.768} C_DIS
LIN {X -0.087,Y -510.291,Z 998.143,A 0.000,B 0.000,C 90.000,E1 241.719} C_DIS
LIN {X 0.188,Y -507.798,Z 998.135,A 0.000,B 0.000,C 90.000,E1 240.205} C_DIS
LIN {X -0.080,Y -505.678,Z 998.128,A 0.000,B 0.000,C 90.000,E1 239.046} C_DIS
LIN {X 0.103,Y -502.748,Z 998.120,A 0.000,B 0.000,C 90.000,E1 237.533} C_DIS
LIN {X 0.043,Y -500.270,Z 998.113,A 0.000,B 0.000,C 90.000,E1 236.342} C_DIS
LIN {X -0.196,Y -498.271,Z 998.108,A 0.000,B 0.000,C 90.000,E1 235.468} C_DIS
LIN {X -0.181,Y -496.230,Z 998.103,A 0.000,B 0.000,C 90.000,E1 234.562} C_DIS
LIN {X 0.101,Y -494.030,Z 998.098,A 0.000,B 0.000,C 90.000,E1 233.623} C_DIS
LIN {X -0.249,Y -488.809,Z 998.086,A 0.000,B 0.000,C 90.000,E1 231.537} C_DIS
LIN {X 0.089,Y -485.917,Z 998.079,A 0.000,B 0.000,C 90.000,E1 230.275} C_DIS
LIN {X -0.043,Y -481.663,Z 998.069,A 0.000,B 0.000,C 90.000,E1 228.447} C_DIS
LIN {X 0.065,Y -475.673,Z 998.054,A 0.000,B 0.000,C 90.000,E1 225.648} C_DIS
LIN {X -0.089,Y -472.427,Z 998.045,A 0.000,B 0.000,C 90.000,E1 224.109} C_DIS
LIN {X 0.032,Y -469.005,Z 998.036,A 0.000,B 0.000,C 90.000,E1 222.528} C_DIS
LIN {X -0.062,Y -464.172,Z 998.024,A 0.000,B 0.000,C 90.000,E1 220.334} C_DIS
LIN {X 0.038,Y -459.849,Z 998.013,A 0.000,B 0.000,C 90.000,E1 218.418} C_DIS
LIN {X 0.030,Y -455.696,Z 998.003,A 0.000,B 0.000,C 90.000,E1 216.503} C_DIS
LIN {X -0.259,Y -451.455,Z 997.992,A 0.000,B 0.000,C 90.000,E1 214.612} C_DIS
LIN {X 0.031,Y -447.976,Z 997.983,A 0.000,B 0.000,C 90.000,E1 212.959} C_DIS
LIN {X 0.070,Y -443.748,Z 997.972,A 0.000,B 0.000,C 90.000,E1 211.003} C_DIS
LIN {X -0.263,Y -440.159,Z 997.963,A 0.000,B 0.000,C 90.000,E1 209.411} C_DIS
LIN {X -0.031,Y -434.194,Z 997.949,A 0.000,B 0.000,C 90.000,E1 206.744} C_DIS
LIN {X 0.012,Y -431.220,Z 997.941,A 0.000,B 0.000,C 90.000,E1 205.412} C_DIS
LIN {X -0.224,Y -425.164,Z 997.926,A 0.000,B 0.000,C 90.000,E1 202.770} C_DIS
LIN {X 0.072,Y -421.435,Z 997.917,A 0.000,B 0.000,C 90.000,E1 201.046} C_DIS
LIN {X -0.246,Y -417.912,Z 997.908,A 0.000,B 0.000,C 90.000,E1 199.396} C_DIS
LIN {X 0.207,Y -412.106,Z 997.891,A 0.000,B 0.000,C 90.000,E1 196.260} C_DIS
LIN {X -0.159,Y -409.096,Z 997.881,A 0.000,B 0.000,C 90.000,E1 194.592} C_DIS
LIN {X 0.094,Y -406.846,Z 997.873,A 0.000,B 0.000,C 90.000,E1 193.175} C_DIS
LIN {X -0.172,Y -403.995,Z 997.864,A 0.000,B 0.000,C 90.000,E1 191.478} C_DIS
LIN {X -0.200,Y -399.113,Z 997.846,A 0.000,B 0.000,C 90.000,E1 188.341} C_DIS
LIN {X 0.164,Y -398.429,Z 997.842,A 0.000,B 0.000,C 90.000,E1 187.587} C_DIS
LIN {X 0.122,Y -398.112,Z 997.838,A 0.000,B 0.000,C 90.000,E1 186.891} C_DIS
LIN {X 0.053,Y -398.083,Z 997.836,A 0.000,B 0.000,C 90.000,E1 186.549} C_DIS
LIN {X 0.004,Y -398.481,Z 997.833,A 0.000,B 0.000,C 90.000,E1 185.853} C_DIS
LIN {X -0.061,Y -398.911,Z 997.831,A 0.000,B 0.000,C 90.000,E1 185.511} C_DIS
LIN {X -0.096,Y -400.609,Z 997.827,A 0.000,B 0.000,C 90.000,E1 184.821} C_DIS
LIN {X -0.143,Y -402.550,Z 997.824,A 0.000,B 0.000,C 90.000,E1 184.302} C_DIS
LIN {X 0.134,Y -405.077,Z 997.821,A 0.000,B 0.000,C 90.000,E1 183.784} C_DIS
LIN {X 0.097,Y -407.227,Z 997.819,A 0.000,B 0.000,C 90.000,E1 183.440} C_DIS
LIN {X -0.018,Y -413.120,Z 997.815,A 0.000,B 0.000,C 90.000,E1 182.694} C_DIS
LIN {X -0.010,Y -420.147,Z 997.811,A 0.000,B 0.000,C 90.000,E1 181.892} C_DIS
LIN {X 0.019,Y -430.162,Z 997.805,A 0.000,B 0.000,C 90.000,E1 180.802} C_DIS
LIN {X -0.195,Y -442.901,Z 997.797,A 0.000,B 0.000,C 90.000,E1 179.484} C_DIS
LIN {X 0.030,Y -452.825,Z 997.791,A 0.000,B 0.000,C 90.000,E1 178.396} C_DIS
LIN {X -0.010,Y -462.259,Z 997.785,A 0.000,B 0.000,C 90.000,E1 177.364} C_DIS
LIN {X -0.165,Y -468.865,Z 997.781,A 0.000,B 0.000,C 90.000,E1 176.617} C_DIS
LIN {X -0.102,Y -474.997,Z 997.777,A 0.000,B 0.000,C 90.000,E1 175.869} C_DIS
LIN {X 0.109,Y -482.044,Z 997.772,A 0.000,B 0.000,C 90.000,E1 174.951} C_DIS
LIN {X -0.184,Y -489.913,Z 997.766,A 0.000,B 0.000,C 90.000,E1 173.913} C_DIS
LIN {X 0.110,Y -497.352,Z 997.760,A 0.000,B 0.000,C 90.000,E1 172.818} C_DIS
LIN {X -0.097,Y -506.672,Z 997.753,A 0.000,B 0.000,C 90.000,E1 171.489} C_DIS
LIN {X 0.180,Y -512.697,Z 997.748,A 0.000,B 0.000,C 90.000,E1 170.566} C_DIS
LIN {X -0.096,Y -520.945,Z 997.740,A 0.000,B 0.000,C 90.000,E1 169.275} C_DIS
LIN {X -0.221,Y -530.729,Z 997.732,A 0.000,B 0.000,C 90.000,E1 167.701} C_DIS
LIN {X 0.135,Y -539.239,Z 997.724,A 0.000,B 0.000,C 90.000,E1 166.228} C_DIS
LIN {X 0.038,Y -545.830,Z 997.717,A 0.000,B 0.000,C 90.000,E1 165.102} C_DIS
LIN {X 0.172,Y -551.572,Z 997.712,A 0.000,B 0.000,C 90.000,E1 164.102} C_DIS
LIN {X 0.116,Y -558.501,Z 997.705,A 0.000,B 0.000,C 90.000,E1 162.851} C_DIS
LIN {X 0.228,Y -565.910,Z 997.697,A 0.000,B 0.000,C 90.000,E1 161.456} C_DIS
LIN {X 0.033,Y -572.298,Z 997.690,A 0.000,B 0.000,C 90.000,E1 160.242} C_DIS
LIN {X -0.149,Y -578.949,Z 997.683,A 0.000,B 0.000,C 90.000,E1 158.901} C_DIS
LIN {X 0.087,Y -581.475,Z 997.680,A 0.000,B 0.000,C 90.000,E1 158.337} C_DIS
LIN {X -0.140,Y -586.262,Z 997.674,A 0.000,B 0.000,C 90.000,E1 157.283} C_DIS
LIN {X 0.229,Y -590.847,Z 997.668,A 0.000,B 0.000,C 90.000,E1 156.177} C_DIS
LIN {X -0.085,Y -594.020,Z 997.663,A 0.000,B 0.000,C 90.000,E1 155.409} C_DIS
LIN {X 0.176,Y -596.893,Z 997.659,A 0.000,B 0.000,C 90.000,E1 154.588} C_DIS
LIN {X -0.070,Y -599.568,Z 997.655,A 0.000,B 0.000,C 90.000,E1 153.819} C_DIS
LIN {X 0.111,Y -603.633,Z 997.647,A 0.000,B 0.000,C 90.000,E1 152.487} C_DIS
LIN {X 0.157,Y -606.748,Z 997.641,A 0.000,B 0.000,C 90.000,E1 151.435} C_DIS
LIN {X 0.161,Y -611.294,Z 997.633,A 0.000,B 0.000,C 90.000,E1 149.871} C_DIS
LIN {X 0.030,Y -615.669,Z 997.624,A 0.000,B 0.000,C 90.000,E1 148.329} C_DIS
LIN {X -0.020,Y -619.832,Z 997.616,A 0.000,B 0.000,C 90.000,E1 146.786} C_DIS
LIN {X -0.011,Y -625.560,Z 997.604,A 0.000,B 0.000,C 90.000,E1 144.736} C_DIS
LIN {X -0.025,Y -629.076,Z 997.597,A 0.000,B 0.000,C 90.000,E1 143.463} C_DIS
LIN {X 0.381,Y -633.302,Z 997.589,A 0.000,B 0.000,C 90.000,E1 141.904} C_DIS
LIN {X -0.138,Y -637.400,Z 997.580,A 0.000,B 0.000,C 90.000,E1 140.436} C_DIS
LIN {X -0.081,Y -640.766,Z 997.573,A 0.000,B 0.000,C 90.000,E1 139.175} C_DIS
LIN {X -0.028,Y -644.065,Z 997.566,A 0.000,B 0.000,C 90.000,E1 137.919} C_DIS
LIN {X 0.322,Y -650.272,Z 997.554,A 0.000,B 0.000,C 90.000,E1 135.648} C_DIS
LIN {X -0.045,Y -656.341,Z 997.543,A 0.000,B 0.000,C 90.000,E1 133.704} C_DIS
LIN {X -0.235,Y -662.874,Z 997.532,A 0.000,B 0.000,C 90.000,E1 131.757} C_DIS
LIN {X -0.249,Y -667.090,Z 997.525,A 0.000,B 0.000,C 90.000,E1 130.539} C_DIS
LIN {X 0.318,Y -671.121,Z 997.518,A 0.000,B 0.000,C 90.000,E1 129.277} C_DIS
LIN {X 0.008,Y -674.794,Z 997.512,A 0.000,B 0.000,C 90.000,E1 128.096} C_DIS
LIN {X -0.114,Y -679.053,Z 997.504,A 0.000,B 0.000,C 90.000,E1 126.664} C_DIS
LIN {X -0.157,Y -683.107,Z 997.496,A 0.000,B 0.000,C 90.000,E1 125.231} C_DIS
LIN {X -0.155,Y -686.424,Z 997.489,A 0.000,B 0.000,C 90.000,E1 124.040} C_DIS
LIN {X 0.093,Y -689.437,Z 997.482,A 0.000,B 0.000,C 90.000,E1 122.832} C_DIS
LIN {X 0.049,Y -693.106,Z 997.475,A 0.000,B 0.000,C 90.000,E1 121.416} C_DIS
LIN {X -0.179,Y -695.977,Z 997.468,A 0.000,B 0.000,C 90.000,E1 120.256} C_DIS
LIN {X 0.229,Y -697.830,Z 997.463,A 0.000,B 0.000,C 90.000,E1 119.283} C_DIS
LIN {X -0.209,Y -698.972,Z 997.459,A 0.000,B 0.000,C 90.000,E1 118.615} C_DIS
LIN {X 0.241,Y -700.112,Z 997.454,A 0.000,B 0.000,C 90.000,E1 117.641} C_DIS
LIN {X -0.045,Y -701.469,Z 997.445,A 0.000,B 0.000,C 90.000,E1 116.027} C_DIS
LIN {X -0.156,Y -702.023,Z 997.441,A 0.000,B 0.000,C 90.000,E1 115.335} C_DIS
LIN {X 0.019,Y -702.372,Z 997.436,A 0.000,B 0.000,C 90.000,E1 114.387} C_DIS
LIN {X 0.008,Y -702.379,Z 997.434,A 0.000,B 0.000,C 90.000,E1 114.155} C_DIS
LIN {X -0.081,Y -701.849,Z 997.432,A 0.000,B 0.000,C 90.000,E1 113.695} C_DIS
LIN {X -0.087,Y -701.366,Z 997.430,A 0.000,B 0.000,C 90.000,E1 113.462} C_DIS
LIN {X -0.329,Y -698.622,Z 997.427,A 0.000,B 0.000,C 90.000,E1 112.898} C_DIS
LIN {X -0.195,Y -697.737,Z 997.426,A 0.000,B 0.000,C 90.000,E1 112.770} C_DIS
LIN {X 0.039,Y -693.765,Z 997.425,A 0.000,B 0.000,C 90.000,E1 112.408} C_DIS
LIN {X -0.064,Y -690.874,Z 997.423,A 0.000,B 0.000,C 90.000,E1 112.206} C_DIS
LIN {X 0.231,Y -688.494,Z 997.423,A 0.000,B 0.000,C 90.000,E1 112.078} C_DIS
LIN {X -0.195,Y -684.379,Z 997.422,A 0.000,B 0.000,C 90.000,E1 111.972} C_DIS
LIN {X -0.361,Y -675.807,Z 997.421,A 0.000,B 0.000,C 90.000,E1 111.844} C_DIS
LIN {X 0.163,Y -674.895,Z 997.421,A 0.000,B 0.000,C 90.000,E1 111.791} C_DIS
LIN {X 0.102,Y -619.560,Z 997.421,A 0.000,B 0.000,C 90.000,E1 111.791} C_DIS
LIN {X -0.220,Y -616.729,Z 997.421,A 0.000,B 0.000,C 90.000,E1 111.770} C_DIS
LIN {X -0.169,Y -610.359,Z 997.420,A 0.000,B 0.000,C 90.000,E1 111.589} C_DIS
LIN {X -0.240,Y -602.613,Z 997.418,A 0.000,B 0.000,C 90.000,E1 111.280} C_DIS
LIN {X 0.147,Y -601.071,Z 997.418,A 0.000,B 0.000,C 90.000,E1 111.173} C_DIS
LIN {X 0.291,Y -594.672,Z 997.416,A 0.000,B 0.000,C 90.000,E1 110.791} C_DIS
LIN {X -0.131,Y -590.421,Z 997.414,A 0.000,B 0.000,C 90.000,E1 110.536} C_DIS
LIN {X 0.029,Y -576.945,Z 997.408,A 0.000,B 0.000,C 90.000,E1 109.450} C_DIS
LIN {X 0.279,Y -572.592,Z 997.406,A 0.000,B 0.000,C 90.000,E1 109.087} C_DIS
LIN {X 0.264,Y -564.228,Z 997.404,A 0.000,B 0.000,C 90.000,E1 108.598} C_DIS
LIN {X 0.188,Y -551.040,Z 997.400,A 0.000,B 0.000,C 90.000,E1 107.946} C_DIS
LIN {X 0.110,Y -550.093,Z 997.399,A 0.000,B 0.000,C 90.000,E1 107.873} C_DIS
LIN {X 0.056,Y -549.051,Z 997.399,A 0.000,B 0.000,C 90.000,E1 107.764} C_DIS
LIN {X 0.014,Y -549.030,Z 997.399,A 0.000,B 0.000,C 90.000,E1 107.764} C_DIS
LIN {X 0.162,Y -548.632,Z 997.397,A 0.000,B 0.000,C 90.000,E1 107.511} C_DIS
LIN {X -0.181,Y -548.598,Z 997.394,A 0.000,B 0.000,C 90.000,E1 106.985} C_DIS
LIN {X -0.016,Y -549.107,Z 997.388,A 0.000,B 0.000,C 90.000,E1 105.843} C_DIS
LIN {X -0.077,Y -550.066,Z 997.377,A 0.000,B 0.000,C 90.000,E1 103.883} C_DIS
LIN {X 0.034,Y -553.617,Z 997.354,A 0.000,B 0.000,C 90.000,E1 99.670} C_DIS
LIN {X 0.058,Y -555.419,Z 997.344,A 0.000,B 0.000,C 90.000,E1 97.992} C_DIS
LIN {X -0.064,Y -556.621,Z 997.338,A 0.000,B 0.000,C 90.000,E1 96.891} C_DIS
LIN {X -0.240,Y -557.659,Z 997.332,A 0.000,B 0.000,C 90.000,E1 95.796} C_DIS
LIN {X 0.152,Y -558.487,Z 997.326,A 0.000,B 0.000,C 90.000,E1 94.645} C_DIS
LIN {X 0.041,Y -559.381,Z 997.318,A 0.000,B 0.000,C 90.000,E1 93.269} C_DIS
LIN {X -0.044,Y -560.096,Z 997.311,A 0.000,B 0.000,C 90.000,E1 91.892} C_DIS
LIN {X 0.069,Y -561.076,Z 997.300,A 0.000,B 0.000,C 90.000,E1 89.943} C_DIS
LIN {X -0.105,Y -561.566,Z 997.294,A 0.000,B 0.000,C 90.000,E1 88.854} C_DIS
LIN {X -0.161,Y -561.901,Z 997.286,A 0.000,B 0.000,C 90.000,E1 87.478} C_DIS
LIN {X -0.079,Y -562.175,Z 997.277,A 0.000,B 0.000,C 90.000,E1 85.812} C_DIS
LIN {X 0.149,Y -562.435,Z 997.266,A 0.000,B 0.000,C 90.000,E1 83.856} C_DIS
LIN {X -0.119,Y -562.813,Z 997.255,A 0.000,B 0.000,C 90.000,E1 81.951} C_DIS
LIN {X 0.252,Y -563.341,Z 997.245,A 0.000,B 0.000,C 90.000,E1 79.982} C_DIS
LIN {X 0.118,Y -564.075,Z 997.235,A 0.000,B 0.000,C 90.000,E1 78.342} C_DIS
LIN {X 0.007,Y -564.929,Z 997.226,A 0.000,B 0.000,C 90.000,E1 76.700} C_DIS
LIN {X -0.178,Y -566.384,Z 997.214,A 0.000,B 0.000,C 90.000,E1 74.519} C_DIS
LIN {X -0.188,Y -567.771,Z 997.203,A 0.000,B 0.000,C 90.000,E1 72.598} C_DIS
LIN {X -0.121,Y -568.771,Z 997.196,A 0.000,B 0.000,C 90.000,E1 71.221} C_DIS
LIN {X 0.139,Y -569.662,Z 997.188,A 0.000,B 0.000,C 90.000,E1 69.826} C_DIS
LIN {X 0.081,Y -570.454,Z 997.180,A 0.000,B 0.000,C 90.000,E1 68.465} C_DIS
LIN {X -0.125,Y -571.279,Z 997.171,A 0.000,B 0.000,C 90.000,E1 66.847} C_DIS
LIN {X 0.015,Y -571.748,Z 997.165,A 0.000,B 0.000,C 90.000,E1 65.741} C_DIS
LIN {X -0.298,Y -572.291,Z 997.158,A 0.000,B 0.000,C 90.000,E1 64.409} C_DIS
LIN {X 0.167,Y -572.729,Z 997.150,A 0.000,B 0.000,C 90.000,E1 62.999} C_DIS
LIN {X -0.031,Y -573.166,Z 997.141,A 0.000,B 0.000,C 90.000,E1 61.385} C_DIS
LIN {X 0.050,Y -573.571,Z 997.132,A 0.000,B 0.000,C 90.000,E1 59.744} C_DIS
LIN {X -0.195,Y -573.788,Z 997.124,A 0.000,B 0.000,C 90.000,E1 58.408} C_DIS
LIN {X 0.008,Y -574.002,Z 997.115,A 0.000,B 0.000,C 90.000,E1 56.755} C_DIS
LIN {X 0.079,Y -574.156,Z 997.108,A 0.000,B 0.000,C 90.000,E1 55.388} C_DIS
LIN {X -0.139,Y -574.090,Z 997.102,A 0.000,B 0.000,C 90.000,E1 54.322} C_DIS
LIN {X -0.041,Y -574.007,Z 997.097,A 0.000,B 0.000,C 90.000,E1 53.497} C_DIS
LIN {X -0.063,Y -573.781,Z 997.093,A 0.000,B 0.000,C 90.000,E1 52.683} C_DIS
LIN {X -0.291,Y -573.221,Z 997.087,A 0.000,B 0.000,C 90.000,E1 51.618} C_DIS
LIN {X -0.178,Y -572.578,Z 997.081,A 0.000,B 0.000,C 90.000,E1 50.517} C_DIS
LIN {X 0.293,Y -571.730,Z 997.075,A 0.000,B 0.000,C 90.000,E1 49.380} C_DIS
LIN {X -0.055,Y -570.703,Z 997.068,A 0.000,B 0.000,C 90.000,E1 48.324} C_DIS
LIN {X 0.267,Y -569.779,Z 997.064,A 0.000,B 0.000,C 90.000,E1 47.472} C_DIS
LIN {X 0.077,Y -569.096,Z 997.061,A 0.000,B 0.000,C 90.000,E1 46.944} C_DIS
LIN {X -0.342,Y -567.350,Z 997.055,A 0.000,B 0.000,C 90.000,E1 45.891} C_DIS
LIN {X -0.065,Y -565.837,Z 997.050,A 0.000,B 0.000,C 90.000,E1 45.040} C_DIS
LIN {X -0.122,Y -563.553,Z 997.044,A 0.000,B 0.000,C 90.000,E1 43.947} C_DIS
LIN {X 0.120,Y -561.563,Z 997.040,A 0.000,B 0.000,C 90.000,E1 43.095} C_DIS
LIN {X -0.072,Y -559.277,Z 997.035,A 0.000,B 0.000,C 90.000,E1 42.285} C_DIS
LIN {X 0.196,Y -555.841,Z 997.029,A 0.000,B 0.000,C 90.000,E1 41.148} C_DIS
LIN {X -0.010,Y -552.850,Z 997.024,A 0.000,B 0.000,C 90.000,E1 40.334} C_DIS
LIN {X 0.050,Y -550.690,Z 997.021,A 0.000,B 0.000,C 90.000,E1 39.769} C_DIS
LIN {X 0.017,Y -547.714,Z 997.017,A 0.000,B 0.000,C 90.000,E1 39.072} C_DIS
LIN {X -0.120,Y -544.542,Z 997.013,A 0.000,B 0.000,C 90.000,E1 38.382} C_DIS
LIN {X 0.156,Y -539.832,Z 997.008,A 0.000,B 0.000,C 90.000,E1 37.363} C_DIS
LIN {X 0.205,Y -533.936,Z 997.001,A 0.000,B 0.000,C 90.000,E1 36.217} C_DIS
LIN {X -0.123,Y -529.215,Z 996.997,A 0.000,B 0.000,C 90.000,E1 35.391} C_DIS
LIN {X -0.163,Y -525.873,Z 996.993,A 0.000,B 0.000,C 90.000,E1 34.818} C_DIS
LIN {X -0.012,Y -519.648,Z 996.988,A 0.000,B 0.000,C 90.000,E1 33.785} C_DIS
LIN {X -0.130,Y -515.892,Z 996.984,A 0.000,B 0.000,C 90.000,E1 33.214} C_DIS
LIN {X -0.123,Y -511.847,Z 996.981,A 0.000,B 0.000,C 90.000,E1 32.625} C_DIS
LIN {X 0.130,Y -507.623,Z 996.978,A 0.000,B 0.000,C 90.000,E1 32.005} C_DIS
LIN {X 0.082,Y -503.050,Z 996.975,A 0.000,B 0.000,C 90.000,E1 31.416} C_DIS
LIN {X 0.261,Y -498.156,Z 996.971,A 0.000,B 0.000,C 90.000,E1 30.797} C_DIS
LIN {X -0.075,Y -494.238,Z 996.969,A 0.000,B 0.000,C 90.000,E1 30.384} C_DIS
LIN {X 0.074,Y -486.098,Z 996.964,A 0.000,B 0.000,C 90.000,E1 29.489} C_DIS
LIN {X 0.270,Y -476.109,Z 996.958,A 0.000,B 0.000,C 90.000,E1 28.487} C_DIS
LIN {X -0.218,Y -467.364,Z 996.954,A 0.000,B 0.000,C 90.000,E1 27.719} C_DIS
LIN {X 0.170,Y -461.479,Z 996.951,A 0.000,B 0.000,C 90.000,E1 27.129} C_DIS
LIN {X -0.001,Y -455.345,Z 996.948,A 0.000,B 0.000,C 90.000,E1 26.616} C_DIS
LIN {X 0.046,Y -446.461,Z 996.944,A 0.000,B 0.000,C 90.000,E1 25.848} C_DIS
LIN {X 0.233,Y -434.290,Z 996.938,A 0.000,B 0.000,C 90.000,E1 24.771} C_DIS
LIN {X -0.159,Y -419.457,Z 996.930,A 0.000,B 0.000,C 90.000,E1 23.462} C_DIS
LIN {X -0.229,Y -406.454,Z 996.923,A 0.000,B 0.000,C 90.000,E1 22.153} C_DIS
LIN {X -0.130,Y -399.401,Z 996.919,A 0.000,B 0.000,C 90.000,E1 21.354} C_DIS
LIN {X 0.195,Y -396.638,Z 996.917,A 0.000,B 0.000,C 90.000,E1 20.972} C_DIS
LIN {X 0.137,Y -392.948,Z 996.913,A 0.000,B 0.000,C 90.000,E1 20.375} C_DIS
LIN {X -0.214,Y -391.130,Z 996.911,A 0.000,B 0.000,C 90.000,E1 19.939} C_DIS
LIN {X 0.160,Y -390.408,Z 996.908,A 0.000,B 0.000,C 90.000,E1 19.396} C_DIS
LIN {X 0.052,Y -390.244,Z 996.907,A 0.000,B 0.000,C 90.000,E1 19.322} C_DIS
LIN {X 0.107,Y -390.479,Z 996.902,A 0.000,B 0.000,C 90.000,E1 18.417} C_DIS
LIN {X -0.133,Y -393.945,Z 996.883,A 0.000,B 0.000,C 90.000,E1 14.898} C_DIS
LIN {X -0.071,Y -399.039,Z 996.861,A 0.000,B 0.000,C 90.000,E1 11.007} C_DIS
LIN {X 0.178,Y -405.575,Z 996.840,A 0.000,B 0.000,C 90.000,E1 7.125} C_DIS
LIN {X 0.160,Y -412.675,Z 996.821,A 0.000,B 0.000,C 90.000,E1 3.669} C_DIS
LIN {X -0.210,Y -416.427,Z 996.811,A 0.000,B 0.000,C 90.000,E1 2.007} C_DIS
LIN {X -0.182,Y -417.185,Z 996.809,A 0.000,B 0.000,C 90.000,E1 1.661} C_DIS
LIN {X -0.091,Y -419.436,Z 996.805,A 0.000,B 0.000,C 90.000,E1 0.974} C_DIS
LIN {X -0.047,Y -421.942,Z 996.803,A 0.000,B 0.000,C 90.000,E1 0.458} C_DIS
LIN {X -0.129,Y -423.439,Z 996.801,A 0.000,B 0.000,C 90.000,E1 0.229} C_DIS
LIN {X 0.046,Y -428.419,Z 996.799,A 0.000,B 0.000,C 90.000,E1 359.714} C_DIS
LIN {X 0.200,Y -433.300,Z 996.797,A 0.000,B 0.000,C 90.000,E1 359.370} C_DIS
LIN {X -0.163,Y -452.489,Z 996.791,A 0.000,B 0.000,C 90.000,E1 358.339} C_DIS
LIN {X -0.087,Y -467.289,Z 996.786,A 0.000,B 0.000,C 90.000,E1 357.478} C_DIS
LIN {X 0.104,Y -484.048,Z 996.781,A 0.000,B 0.000,C 90.000,E1 356.502} C_DIS
LIN {X 0.006,Y -492.199,Z 996.778,A 0.000,B 0.000,C 90.000,E1 356.045} C_DIS
LIN {X -0.037,Y -501.991,Z 996.775,A 0.000,B 0.000,C 90.000,E1 355.469} C_DIS
LIN {X 0.119,Y -509.979,Z 996.772,A 0.000,B 0.000,C 90.000,E1 354.951} C_DIS
LIN {X -0.243,Y -518.957,Z 996.769,A 0.000,B 0.000,C 90.000,E1 354.375} C_DIS
LIN {X -0.021,Y -527.975,Z 996.765,A 0.000,B 0.000,C 90.000,E1 353.685} C_DIS
LIN {X -0.066,Y -533.813,Z 996.762,A 0.000,B 0.000,C 90.000,E1 353.223} C_DIS
LIN {X -0.100,Y -539.154,Z 996.760,A 0.000,B 0.000,C 90.000,E1 352.761} C_DIS
LIN {X 0.132,Y -543.245,Z 996.758,A 0.000,B 0.000,C 90.000,E1 352.356} C_DIS
LIN {X -0.126,Y -549.792,Z 996.754,A 0.000,B 0.000,C 90.000,E1 351.724} C_DIS
LIN {X -0.240,Y -554.787,Z 996.751,A 0.000,B 0.000,C 90.000,E1 351.197} C_DIS
LIN {X 0.160,Y -559.263,Z 996.748,A 0.000,B 0.000,C 90.000,E1 350.622} C_DIS
LIN {X -0.104,Y -563.620,Z 996.745,A 0.000,B 0.000,C 90.000,E1 350.095} C_DIS
LIN {X 0.222,Y -567.530,Z 996.742,A 0.000,B 0.000,C 90.000,E1 349.511} C_DIS
LIN {X -0.087,Y -571.112,Z 996.739,A 0.000,B 0.000,C 90.000,E1 348.993} C_DIS
LIN {X -0.188,Y -576.759,Z 996.734,A 0.000,B 0.000,C 90.000,E1 348.049} C_DIS
LIN {X 0.122,Y -582.526,Z 996.728,A 0.000,B 0.000,C 90.000,E1 346.937} C_DIS
LIN {X 0.172,Y -587.321,Z 996.722,A 0.000,B 0.000,C 90.000,E1 345.992} C_DIS
LIN {X -0.102,Y -593.733,Z 996.715,A 0.000,B 0.000,C 90.000,E1 344.685} C_DIS
LIN {X 0.144,Y -597.357,Z 996.711,A 0.000,B 0.000,C 90.000,E1 343.866} C_DIS
LIN {X 0.009,Y -600.736,Z 996.706,A 0.000,B 0.000,C 90.000,E1 343.087} C_DIS
LIN {X -0.188,Y -605.071,Z 996.700,A 0.000,B 0.000,C 90.000,E1 342.054} C_DIS
LIN {X -0.244,Y -608.301,Z 996.696,A 0.000,B 0.000,C 90.000,E1 341.275} C_DIS
LIN {X 0.189,Y -613.200,Z 996.689,A 0.000,B 0.000,C 90.000,E1 339.934} C_DIS
LIN {X -0.115,Y -614.992,Z 996.686,A 0.000,B 0.000,C 90.000,E1 339.444} C_DIS
LIN {X -0.163,Y -619.894,Z 996.677,A 0.000,B 0.000,C 90.000,E1 337.901} C_DIS
LIN {X -0.117,Y -623.671,Z 996.670,A 0.000,B 0.000,C 90.000,E1 336.613} C_DIS
LIN {X -0.355,Y -626.516,Z 996.664,A 0.000,B 0.000,C 90.000,E1 335.613} C_DIS
LIN {X 0.258,Y -628.473,Z 996.660,A 0.000,B 0.000,C 90.000,E1 334.793} C_DIS
LIN {X 0.352,Y -630.964,Z 996.654,A 0.000,B 0.000,C 90.000,E1 333.768} C_DIS
LIN {X -0.117,Y -632.588,Z 996.650,A 0.000,B 0.000,C 90.000,E1 333.050} C_DIS
LIN {X 0.163,Y -636.131,Z 996.640,A 0.000,B 0.000,C 90.000,E1 331.257} C_DIS
LIN {X 0.155,Y -638.443,Z 996.633,A 0.000,B 0.000,C 90.000,E1 329.999} C_DIS
LIN {X 0.185,Y -640.440,Z 996.626,A 0.000,B 0.000,C 90.000,E1 328.742} C_DIS
LIN {X 0.132,Y -641.567,Z 996.622,A 0.000,B 0.000,C 90.000,E1 327.995} C_DIS
LIN {X 0.059,Y -643.384,Z 996.614,A 0.000,B 0.000,C 90.000,E1 326.501} C_DIS
LIN {X -0.088,Y -644.422,Z 996.608,A 0.000,B 0.000,C 90.000,E1 325.515} C_DIS
